IF VisitingExtension.Alarms.HasAlarms THEN
	serializer.addkey('alarms');
	serializer.StartArray();
	VisitingExtension.Alarms.Accept(THIS^);
	serializer.EndArray();
END_IF

IF VisitingExtension.InputPorts.HasInputPorts THEN
	serializer.addkey('inputPorts');
	serializer.StartArray();
	VisitingExtension.InputPorts.Accept(THIS^);
	serializer.EndArray();
END_IF

IF VisitingExtension.OutputPorts.HasOutputPorts THEN
	serializer.addkey('outputPorts');
	serializer.StartArray();
	VisitingExtension.OutputPorts.Accept(THIS^);
	serializer.EndArray();
END_IF

IF VisitingExtension.Parameters.HasParameters THEN
	serializer.addkey('parameters');
	serializer.StartArray();
	VisitingExtension.Parameters.Accept(THIS^);
	serializer.EndArray();
END_IF

IF VisitingExtension.Contents.HasContents THEN
	serializer.addkey('contents');
	serializer.StartArray();
	VisitingExtension.Contents.Accept(THIS^);
	serializer.EndArray();
END_IF

Serializer.EndObject();
END_METHOD

METHOD VisitInputPort
VAR_INPUT
	VisitingInputPort : I_InputPort;
END_VAR
serializer.StartObject();

serializer.AddKeyString('name', VisitingInputPort.Name);
serializer.Addkey('datatype');
VisitingInputPort.Data.SerializeTypeWith(serializer);

IF VisitingInputPort.Metadatum.HasMetadata THEN
	serializer.addkey('metadata');
	serializer.StartArray();
	VisitingInputPort.Metadatum.Accept(THIS^);
	serializer.EndArray();
END_IF

serializer.EndObject();
END_METHOD

METHOD VisitMetadatum
VAR_INPUT
	VisitingMetadatum : I_Metadata;
END_VAR
serializer.StartObject();
serializer.AddKeyString('name', VisitingMetadatum.Name);
serializer.AddkeyObject('value', VisitingMetadatum.Data);
serializer.EndObject();
END_METHOD

METHOD VisitNode
VAR_INPUT
	VisitingNode : I_Node;
END_VAR
serializer.StartObject();

IF VisitingNode.Metadatum.HasMetadata THEN
	serializer.addkey('metadata');
	serializer.StartArray();
	VisitingNode.Metadatum.Accept(THIS^);
	serializer.EndArray();
END_IF

IF VisitingNode.Alarms.HasAlarms THEN
	serializer.addkey('alarms');
	serializer.StartArray();
	VisitingNode.Alarms.Accept(THIS^);
	serializer.EndArray();
END_IF

IF VisitingNode.Extensions.HasExtensions THEN
	serializer.addkey('extensions');
	serializer.StartArray();
	VisitingNode.Extensions.Accept(THIS^);
	serializer.EndArray();
END_IF

IF VisitingNode.InputPorts.HasInputPorts THEN
	serializer.addkey('inputPorts');
	serializer.StartArray();
	VisitingNode.InputPorts.Accept(THIS^);
	serializer.EndArray();
END_IF

IF VisitingNode.OutputPorts.HasOutputPorts THEN
	serializer.addkey('outputPorts');
	serializer.StartArray();
	VisitingNode.OutputPorts.Accept(THIS^);
	serializer.EndArray();
END_IF

IF VisitingNode.Parameters.HasParameters THEN
	serializer.addkey('parameters');
	serializer.StartArray();
	VisitingNode.Parameters.Accept(THIS^);
	serializer.EndArray();
END_IF

IF VisitingNode.Contents.HasContents THEN
	serializer.addkey('contents');
	serializer.StartArray();
	VisitingNode.Contents.Accept(THIS^);
	serializer.EndArray();
END_IF

serializer.EndObject();
END_METHOD

METHOD VisitNodeFactory
VAR_INPUT
	VisitingNodeFactory : I_NodeFactory;
END_VAR
serializer.StartObject();
serializer.AddKey('blueprints');
serializer.StartArray();
VisitingNodeFactory.NodePrototypes.Accept(THIS^);
serializer.EndArray();
serializer.AddKeyUdint('returnedCount', blueprintsCollected);
serializer.AddKeyUdint('totalCount', totalBlueprints);
serializer.AddKeyUdint('nextOffset', offset + blueprintsCollected);
serializer.AddKeyBool('hasMore', offset + blueprintsCollected < totalBlueprints); 
serializer.EndObject();
END_METHOD

METHOD VisitNodePrototype
VAR_INPUT
	VisitingPrototype : I_NodePrototype;
END_VAR
// we're not yet in range of collection
IF currentIndex < offset THEN
	currentIndex := currentIndex + 1;
	totalBlueprints := totalBlueprints + 1;
	RETURN;
END_IF

// we're over range of the collection
IF currentIndex > endIndex THEN
	currentIndex := currentIndex + 1;
	totalBlueprints := totalBlueprints + 1;
	RETURN;
END_IF

// we're in the range to collect. 

blueprintsCollected := blueprintsCollected + 1;
currentIndex := currentIndex + 1;
totalBlueprints := totalBlueprints + 1;

serializer.StartObject();
serializer.AddKeyString('path', VisitingPrototype.Path);
serializer.AddKey('node');
VisitingPrototype.Node.Accept(THIS^);
serializer.EndObject();
END_METHOD

METHOD VisitOutputPort
VAR_INPUT
	VisitingOutputPort : I_OutputPort;
END_VAR
serializer.StartObject();

serializer.AddKeyString('name', VisitingOutputPort.Name);
serializer.Addkey('datatype');
VisitingOutputPort.Data.SerializeTypeWith(serializer);

IF VisitingOutputPort.Metadatum.HasMetadata THEN
	serializer.addkey('metadata');
	serializer.StartArray();
	VisitingOutputPort.Metadatum.Accept(THIS^);
	serializer.EndArray();
END_IF

serializer.EndObject();
END_METHOD

METHOD VisitParameter
VAR_INPUT
	VisitingProperty : I_Parameter;
END_VAR
serializer.StartObject();

serializer.AddKeyString('name', VisitingProperty.Name);
serializer.Addkey('datatype');
VisitingProperty.Data.SerializeTypeWith(serializer);
serializer.Addkey('defaultValue');
VisitingProperty.Data.SerializeWith(serializer);

IF VisitingProperty.Metadatum.HasMetadata THEN
	serializer.addkey('metadata');
	serializer.StartArray();
	VisitingProperty.Metadatum.Accept(THIS^);
	serializer.EndArray();
END_IF

Serializer.EndObject();
END_METHOD

END_FUNCTION_BLOCK

// API/Visitors/GetBlueprintsVisitor
{attribute 'linkalways'} 
{attribute 'no_explicit_call' := 'This FB is a CLASS and must be accessed using methods or properties'}
{attribute 'enable_dynamic_creation'}
FUNCTION_BLOCK GetBlueprintsVisitor IMPLEMENTS I_NodeFactoryVisitor, I_NodePrototypeVisitor, I_NodeVisitor, I_ExtensionVisitor, I_InputPortVisitor, I_OutputPortVisitor, I_MetadataVisitor, I_ContentVisitor, I_ParameterVisitor, I_AlarmVisitor
VAR
	serializer : I_Serializer;
END_VAR

METHOD PUBLIC Initialize
VAR_INPUT
	Serializer : I_Serializer;
END_VAR
THIS^.serializer := Serializer;
END_METHOD

METHOD VisitAlarm
VAR_INPUT
	VisitingAlarm : I_Alarm;
END_VAR
serializer.AddString(VisitingAlarm.Message);
END_METHOD

METHOD VisitContent
VAR_INPUT
	VisitingContent : I_Content;
END_VAR
serializer.StartObject();

serializer.AddKeyString('name', VisitingContent.Name);
serializer.Addkey('datatype');
VisitingContent.Data.SerializeTypeWith(serializer);

IF VisitingContent.Metadatum.HasMetadata THEN
	serializer.addkey('metadata');
	serializer.StartArray();
	VisitingContent.Metadatum.Accept(THIS^);
	serializer.EndArray();
END_IF

serializer.EndObject();
END_METHOD

METHOD VisitExtension
VAR_INPUT
	VisitingExtension : I_Extension;
END_VAR
Serializer.StartObject();
Serializer.AddKeyString('name', VisitingExtension.Name);

IF VisitingExtension.Metadatum.HasMetadata THEN
	serializer.addkey('metadata');
	serializer.StartArray();
	VisitingExtension.Metadatum.Accept(THIS^);
	serializer.EndArray();
END_IF

IF VisitingExtension.Alarms.HasAlarms THEN
	serializer.addkey('alarms');
	serializer.StartArray();
	VisitingExtension.Alarms.Accept(THIS^);
	serializer.EndArray();
END_IF

IF VisitingExtension.InputPorts.HasInputPorts THEN
	serializer.addkey('inputPorts');
	serializer.StartArray();
	VisitingExtension.InputPorts.Accept(THIS^);
	serializer.EndArray();
END_IF

IF VisitingExtension.OutputPorts.HasOutputPorts THEN
	serializer.addkey('outputPorts');
	serializer.StartArray();
	VisitingExtension.OutputPorts.Accept(THIS^);
	serializer.EndArray();
END_IF

IF VisitingExtension.Parameters.HasParameters THEN
	serializer.addkey('parameters');
	serializer.StartArray();
	VisitingExtension.Parameters.Accept(THIS^);
	serializer.EndArray();
END_IF

IF VisitingExtension.Contents.HasContents THEN
	serializer.addkey('contents');
	serializer.StartArray();
	VisitingExtension.Contents.Accept(THIS^);
	serializer.EndArray();
END_IF

Serializer.EndObject();
END_METHOD

METHOD VisitInputPort
VAR_INPUT
	VisitingInputPort : I_InputPort;
END_VAR
serializer.StartObject();

serializer.AddKeyString('name', VisitingInputPort.Name);
serializer.Addkey('datatype');
VisitingInputPort.Data.SerializeTypeWith(serializer);

IF VisitingInputPort.Metadatum.HasMetadata THEN
	serializer.addkey('metadata');
	serializer.StartArray();
	VisitingInputPort.Metadatum.Accept(THIS^);
	serializer.EndArray();
END_IF

serializer.EndObject();
END_METHOD

METHOD VisitMetadatum
VAR_INPUT
	VisitingMetadatum : I_Metadata;
END_VAR
serializer.StartObject();
serializer.AddKeyString('name', VisitingMetadatum.Name);
serializer.AddkeyObject('value', VisitingMetadatum.Data);
serializer.EndObject();
END_METHOD

METHOD VisitNode
VAR_INPUT
	VisitingNode : I_Node;
END_VAR
serializer.StartObject();

IF VisitingNode.Metadatum.HasMetadata THEN
	serializer.addkey('metadata');
	serializer.StartArray();
	VisitingNode.Metadatum.Accept(THIS^);
	serializer.EndArray();
END_IF

IF VisitingNode.Alarms.HasAlarms THEN
	serializer.addkey('alarms');
	serializer.StartArray();
	VisitingNode.Alarms.Accept(THIS^);
	serializer.EndArray();
END_IF

IF VisitingNode.Extensions.HasExtensions THEN
	serializer.addkey('extensions');
	serializer.StartArray();
	VisitingNode.Extensions.Accept(THIS^);
	serializer.EndArray();
END_IF

IF VisitingNode.InputPorts.HasInputPorts THEN
	serializer.addkey('inputPorts');
	serializer.StartArray();
	VisitingNode.InputPorts.Accept(THIS^);
	serializer.EndArray();
END_IF

IF VisitingNode.OutputPorts.HasOutputPorts THEN
	serializer.addkey('outputPorts');
	serializer.StartArray();
	VisitingNode.OutputPorts.Accept(THIS^);
	serializer.EndArray();
END_IF

IF VisitingNode.Parameters.HasParameters THEN
	serializer.addkey('parameters');
	serializer.StartArray();
	VisitingNode.Parameters.Accept(THIS^);
	serializer.EndArray();
END_IF

IF VisitingNode.Contents.HasContents THEN
	serializer.addkey('contents');
	serializer.StartArray();
	VisitingNode.Contents.Accept(THIS^);
	serializer.EndArray();
END_IF

serializer.EndObject();
END_METHOD

METHOD VisitNodeFactory
VAR_INPUT
	VisitingNodeFactory : I_NodeFactory;
END_VAR
serializer.StartObject();
serializer.AddKey('blueprints');
serializer.StartArray();
VisitingNodeFactory.NodePrototypes.Accept(THIS^);
serializer.EndArray();
serializer.EndObject();
END_METHOD

METHOD VisitNodePrototype
VAR_INPUT
	VisitingPrototype : I_NodePrototype;
END_VAR
serializer.StartObject();
serializer.AddKeyString('path', VisitingPrototype.Path);
serializer.AddKey('node');
VisitingPrototype.Node.Accept(THIS^);
serializer.EndObject();
END_METHOD

METHOD VisitOutputPort
VAR_INPUT
	VisitingOutputPort : I_OutputPort;
END_VAR
serializer.StartObject();

serializer.AddKeyString('name', VisitingOutputPort.Name);
serializer.Addkey('datatype');
VisitingOutputPort.Data.SerializeTypeWith(serializer);

IF VisitingOutputPort.Metadatum.HasMetadata THEN
	serializer.addkey('metadata');
	serializer.StartArray();
	VisitingOutputPort.Metadatum.Accept(THIS^);
	serializer.EndArray();
END_IF

serializer.EndObject();
END_METHOD

METHOD VisitParameter
VAR_INPUT
	VisitingProperty : I_Parameter;
END_VAR
serializer.StartObject();

serializer.AddKeyString('name', VisitingProperty.Name);
serializer.Addkey('datatype');
VisitingProperty.Data.SerializeTypeWith(serializer);
serializer.Addkey('defaultValue');
VisitingProperty.Data.SerializeWith(serializer);

IF VisitingProperty.Metadatum.HasMetadata THEN
	serializer.addkey('metadata');
	serializer.StartArray();
	VisitingProperty.Metadatum.Accept(THIS^);
	serializer.EndArray();
END_IF

Serializer.EndObject();
END_METHOD

END_FUNCTION_BLOCK

// API/Handlers/GetContentValueHandler
{attribute 'linkalways'} 
{attribute 'no_explicit_call' := 'This FB is a CLASS and must be accessed using methods or properties'}
{attribute 'enable_dynamic_creation'}
FUNCTION_BLOCK GetContentValueHandler IMPLEMENTS I_AsynchronousRpcHandler
VAR
	graphRuntimes : I_GraphRuntimeCollection;
END_VAR

METHOD Handle
VAR_INPUT
	Parameters : I_Deserializer;
	Response : I_AsynchronousRpcResponse;
END_VAR
VAR
	runtimeId : T_MAXSTRING;
	graphRuntime : I_GraphRuntime;
	graphInstanceId : T_MAXSTRING;
	graphInstance : I_GraphInstance;
	graphUuid : T_MAXSTRING;
	nodeId : T_MAXSTRING;
	contentName : T_MAXSTRING;
	visitor : RetrieveNodeContentValue;
	serializer : I_Serializer;
	feedback : DeserializerFeedback;
END_VAR
IF graphRuntimes = 0 THEN
	Response.RejectWithError('INTERNAL_ERROR','GetContentValueHandler has not been correctly initialized');
	RETURN;
END_IF

// get runtime
IF Parameters.TryGetKeyString('runtimeId', runtimeId, feedback) THEN
	IF NOT graphRuntimes.TryGetRuntimeById(runtimeId, graphRuntime) THEN
		Response.RejectWithError('INVALID_RUNTIME_ID','The runtimeId is missing or invalid');
		RETURN;
	END_IF
ELSE
	IF NOT graphRuntimes.TryGetDefaultRuntime(graphRuntime) THEN
		Response.RejectWithError('INTERNAL_ERROR','Unable to get default runtime');
		RETURN;
	END_IF
END_IF

// get graph instance
IF Parameters.TryGetKeyString('graphInstanceId', graphInstanceId, feedback) THEN
	IF NOT graphRuntime.TryGetGraphInstance(graphInstanceId, graphInstance) THEN
		Response.RejectWithError('INVALID_GRAPH_INSTANCE_ID','The graphInstanceId is missing or invalid');
		RETURN;
	END_IF
ELSE
	IF NOT graphRuntime.TryGetDefaultGraphInstance(graphInstance) THEN
		Response.RejectWithError('NO_GRAPH_INSTANCE_AVAILABLE','Unable to get default graph instance, i.e. no graph instance is loaded');
		RETURN;
	END_IF
END_IF

// setup the visitor
IF NOT Parameters.TryGetKeyString('graphUuid', graphUuid, feedback) THEN
	Response.RejectWithError('MISSING_GRAPH_UUID_PARAMETER',feedback.FirstError.Message);
	RETURN;
END_IF

IF NOT (graphUuid = graphInstance.Graph.Uuid) THEN
	Response.RejectWithError('GRAPH_UUID_MISSMATCH','The requested uuid did not match the graph instance found');
	RETURN;
END_IF

IF NOT Parameters.TryGetKeyString('nodeId', nodeId, feedback) THEN
	Response.RejectWithError('MISSING_NODE_ID_PARAMETER',feedback.FirstError.Message);
	RETURN;
END_IF

IF NOT Parameters.TryGetKeyString('contentName', contentName, feedback) THEN
	Response.RejectWithError('MISSING_CONTENT_NAME_PARAMETER',feedback.FirstError.Message);
	RETURN;
END_IF

serializer := Response.GetSerializer();
visitor.Initialize(graphUuid, nodeId, contentName, serializer);
graphInstance.graph.Accept(visitor);

IF visitor.Error THEN
	Response.RejectWithError('GET_CONTENT_FAILED',visitor.ErrorMessage);
	serializer.Dispose();
	RETURN;
END_IF

IF NOT visitor.Done THEN
	Response.RejectWithError('GET_CONTENT_FAILED','Unable to get content from graph');
	serializer.Dispose();
	RETURN;
END_IF

Response.CompleteWithSerializer(serializer);
serializer.Dispose();
END_METHOD

METHOD PUBLIC Initialize
VAR_INPUT
	GraphRuntimes : I_GraphRuntimeCollection;
END_VAR
THIS^.graphRuntimes := GraphRuntimes;
END_METHOD

END_FUNCTION_BLOCK

// API/Visitors/RetrieveNodeContentValue
{attribute 'linkalways'} 
{attribute 'no_explicit_call' := 'This FB is a CLASS and must be accessed using methods or properties'}
{attribute 'enable_dynamic_creation'}
FUNCTION_BLOCK RetrieveNodeContentValue IMPLEMENTS I_GraphVisitor, I_NodeVisitor, I_ContentVisitor
VAR
	graphUuid : T_MAXSTRING;
	nodeId : T_MAXSTRING;
	contentName : T_MAXSTRING;
	serializer : I_Serializer;
	_done : BOOL;
	_error : BOOL;
	_errorMessage : T_MAXSTRING;
END_VAR

METHOD PRIVATE LogInvalidContentNameError
VAR_INPUT
END_VAR
_errorMessage := 'Invalid Content Name';
_error := TRUE;
END_METHOD

METHOD PRIVATE LogInvalidNodeIdError
VAR_INPUT
END_VAR
_errorMessage := 'Invalid Node Id';
_error := TRUE;
END_METHOD

METHOD PRIVATE Reset
VAR_INPUT
END_VAR
_done := FALSE;
_errorMessage := '';
_error := FALSE;
END_METHOD

PROPERTY PUBLIC Done : BOOL
GET
Done := _done;
END_GET
END_PROPERTY

PROPERTY PUBLIC Error : BOOL
GET
Error := _error;
END_GET
END_PROPERTY

PROPERTY PUBLIC ErrorMessage : T_MAXSTRING
GET
ErrorMessage := _errorMessage;
END_GET
END_PROPERTY

METHOD PUBLIC Initialize
VAR_INPUT
	GraphUuid : T_MAXSTRING;
	NodeId : T_MAXSTRING;
	ContentName : T_MAXSTRING;
	Serializer : I_Serializer;
END_VAR
THIS^.graphUuid := GraphUuid;
THIS^.nodeId := NodeId;
THIS^.contentName := ContentName;
THIS^.serializer := Serializer;
END_METHOD

METHOD VisitContent
VAR_INPUT
	VisitingContent : I_Content;
END_VAR
VisitingContent.SerializeWith(serializer);
END_METHOD

METHOD VisitGraph
VAR_INPUT
	VisitingGraph : I_Graph;
END_VAR
VAR
	node : I_Node;
END_VAR
Reset();

IF NOT (VisitingGraph.Uuid = graphUuid) THEN
	RETURN;
END_IF

IF NOT VisitingGraph.Nodes.TryGetNodeById(nodeId, node) THEN
	LogInvalidNodeIdError();
	RETURN;
END_IF

node.Accept(THIS^);
END_METHOD

METHOD VisitNode
VAR_INPUT
	VisitingNode : I_Node;
END_VAR
VAR
	content : I_Content;
END_VAR
IF NOT VisitingNode.Contents.TryGetContentByName(contentName, content) THEN
	LogInvalidContentNameError();
	RETURN;
END_IF

content.Accept(THIS^);
END_METHOD

END_FUNCTION_BLOCK

// API/Handlers/GetStatusRpcHandler
{attribute 'linkalways'} 
{attribute 'no_explicit_call' := 'This FB is a CLASS and must be accessed using methods or properties'}
{attribute 'enable_dynamic_creation'}
FUNCTION_BLOCK GetStatusRpcHandler IMPLEMENTS I_AsynchronousRpcHandler
VAR
	graphRuntimes : I_GraphRuntimeCollection;
END_VAR

METHOD Handle
VAR_INPUT
	Parameters : I_Deserializer;
	Response : I_AsynchronousRpcResponse;
END_VAR
VAR
	runtimeId : T_MAXSTRING;
	graphRuntime : I_GraphRuntime;
	graphInstanceId : T_MAXSTRING;
	graphUuid : T_MAXSTRING;
	graphInstance : I_GraphInstance;
	feedback : DeserializerFeedback;
	serializer : I_Serializer;
	getStatusVisitor : GetStatusVisitor;
END_VAR
IF graphRuntimes = 0 THEN
	Response.RejectWithError('INTERNAL_ERROR','GetStatusRpcHandler has not been correctly initialized');
	RETURN;
END_IF

// get runtime
IF Parameters.TryGetKeyString('runtimeId', runtimeId, feedback) THEN
	IF NOT graphRuntimes.TryGetRuntimeById(runtimeId, graphRuntime) THEN
		Response.RejectWithError('INVALID_RUNTIME_ID','The runtimeId is missing or invalid');
		RETURN;
	END_IF
ELSE
	IF NOT graphRuntimes.TryGetDefaultRuntime(graphRuntime) THEN
		Response.RejectWithError('INTERNAL_ERROR','Unable to get default runtime');
		RETURN;
	END_IF
END_IF

// get graph instance
IF Parameters.TryGetKeyString('graphInstanceId', graphInstanceId, feedback) THEN
	IF NOT graphRuntime.TryGetGraphInstance(graphInstanceId, graphInstance) THEN
		Response.RejectWithError('INVALID_GRAPH_INSTANCE_ID','The graphInstanceId is missing or invalid');
		RETURN;
	END_IF
ELSE
	IF NOT graphRuntime.TryGetDefaultGraphInstance(graphInstance) THEN
		Response.RejectWithError('NO_GRAPH_INSTANCE_AVAILABLE','Unable to get default graph instance, i.e. no graph instance is loaded');
		RETURN;
	END_IF
END_IF

// setup the visitor
IF NOT Parameters.TryGetKeyString('graphUuid', graphUuid, feedback) THEN
	Response.RejectWithError('MISSING_GRAPH_UUID_PARAMETER', feedback.FirstError.Message);
	RETURN;
END_IF

IF NOT (graphUuid = graphInstance.Graph.Uuid) THEN
	Response.RejectWithError('GRAPH_UUID_MISSMATCH','The requested uuid did not match the graph instance found');
	RETURN;
END_IF

serializer := Response.GetSerializer();
getStatusVisitor.Initialize(serializer);
getStatusVisitor.VisitGraph(graphInstance.Graph);
Response.CompleteWithSerializer(serializer);
serializer.Dispose();
END_METHOD

METHOD PUBLIC Initialize
VAR_INPUT
	GraphRuntimes : I_GraphRuntimeCollection;
END_VAR
THIS^.graphRuntimes := GraphRuntimes;
END_METHOD

END_FUNCTION_BLOCK

// API/Handlers/UpdateParameterValueHandler
{attribute 'linkalways'} 
{attribute 'no_explicit_call' := 'This FB is a CLASS and must be accessed using methods or properties'}
{attribute 'enable_dynamic_creation'}
FUNCTION_BLOCK UpdateParameterValueHandler IMPLEMENTS I_AsynchronousRpcHandler
VAR
	graphRuntimes : I_GraphRuntimeCollection;
END_VAR

METHOD Handle
VAR_INPUT
	Parameters : I_Deserializer;
	Response : I_AsynchronousRpcResponse;
END_VAR
VAR
	runtimeId : T_MAXSTRING;
	graphRuntime : I_GraphRuntime;
	graphInstanceId : T_MAXSTRING;
	graphUuid : T_MAXSTRING;
	graphInstance : I_GraphInstance;
	nodeId : T_MAXSTRING;
	node : I_Node;
	parameterName : T_MAXSTRING;
	parameter : I_Parameter;
	visitor : RetrieveNodeContentValue;
	serializer : I_Serializer;
	feedback : DeserializerFeedback;
END_VAR
IF graphRuntimes = 0 THEN
	Response.RejectWithError('INTERNAL_ERROR','UpdateParameterValueHandler has not been correctly initialized');
	RETURN;
END_IF

// get runtime
IF Parameters.TryGetKeyString('runtimeId', runtimeId, feedback) THEN
	IF NOT graphRuntimes.TryGetRuntimeById(runtimeId, graphRuntime) THEN
		Response.RejectWithError('INVALID_RUNTIME_ID','The runtimeId is missing or invalid');
		RETURN;
	END_IF
ELSE
	IF NOT graphRuntimes.TryGetDefaultRuntime(graphRuntime) THEN
		Response.RejectWithError('INTERNAL_ERROR','Unable to get default runtime');
		RETURN;
	END_IF
END_IF

// get graph instance
IF Parameters.TryGetKeyString('graphInstanceId', graphInstanceId, feedback) THEN
	IF NOT graphRuntime.TryGetGraphInstance(graphInstanceId, graphInstance) THEN
		Response.RejectWithError('INVALID_GRAPH_INSTANCE_ID','The graphInstanceId is missing or invalid');
		RETURN;
	END_IF
ELSE
	IF NOT graphRuntime.TryGetDefaultGraphInstance(graphInstance) THEN
		Response.RejectWithError('NO_GRAPH_INSTANCE_AVAILABLE','Unable to get default graph instance, i.e. no graph instance is loaded');
		RETURN;
	END_IF
END_IF

// setup the visitor
IF NOT Parameters.TryGetKeyString('graphUuid', graphUuid, feedback) THEN
	Response.RejectWithError('MISSING_GRAPH_UUID_PARAMETER',feedback.FirstError.Message);
	RETURN;
END_IF

IF NOT (graphUuid = graphInstance.Graph.Uuid) THEN
	Response.RejectWithError('GRAPH_UUID_MISSMATCH', 'The requested uuid did not match the graph instance found');
	RETURN;
END_IF

IF NOT Parameters.TryGetKeyString('nodeId', nodeId, feedback) THEN
	Response.RejectWithError('MISSING_NODE_ID_PARAMETER',feedback.FirstError.Message);
	RETURN;
END_IF

IF NOT graphInstance.Graph.Nodes.TryGetNodeById(nodeId, node) THEN
	Response.RejectWithError('INVALID_NODE_ID','Invalid or missing nodeId');
	RETURN;
END_IF

IF NOT Parameters.TryGetKeyString('parameterName', parameterName, feedback) THEN
	Response.RejectWithError('MISSING_PARAMETER_NAME_PARAMETER',feedback.FirstError.Message);
	RETURN;
END_IF

IF NOT node.Parameters.TryGetParameterByName(parameterName, parameter) THEN
	Response.RejectWithError('INVALID_PARAMETER_NAME','Invalid or missing parameterName');
	RETURN;
END_IF

IF NOT Parameters.TryDeserializeKeyToObject ('parameterValue', parameter, feedback) THEN
	Response.RejectWithError('MISSING_PARAMETER_VALUE_PARAMETER',feedback.FirstError.Message);
	RETURN;
END_IF

Response.CompleteWithString(graphUuid);
END_METHOD

METHOD PUBLIC Initialize
VAR_INPUT
	GraphRuntimes : I_GraphRuntimeCollection;
END_VAR
THIS^.graphRuntimes := GraphRuntimes;
END_METHOD

END_FUNCTION_BLOCK

// API/GraphFrameworkApi
{attribute 'linkalways'} 
{attribute 'no_explicit_call' := 'This FB is a CLASS and must be accessed using methods or properties'}
{attribute 'enable_dynamic_creation'}
FUNCTION_BLOCK GraphFrameworkApi IMPLEMENTS I_RpcApi
VAR
	graphFramework : I_GraphFramework;
	graphRuntimes : GraphRuntimeCollection;
	createGraphRpcHandler : CreateGraphRpcHandler;
	getStatusRpcHandler : GetStatusRpcHandler;
	getBlueprintsRpcHandler : GetBlueprintsRpcHandler;
	getContentValueHandler : GetContentValueHandler;
	updateParameterValueHandler : UpdateParameterValueHandler;
END_VAR

METHOD FB_init : BOOL
VAR_INPUT
	bInitRetains : BOOL; // if TRUE, the retain variables are initialized (warm start / cold start)
	bInCopyCode : BOOL;  // if TRUE, the instance afterwards gets moved into the copy code (online change)
	GraphFramework : I_GraphFramework;
	DefaultGraphRuntime : I_GraphRuntime;
END_VAR
THIS^.graphFramework := GraphFramework;
THIS^.graphRuntimes.AddDefaultRuntime(DefaultGraphRuntime);

getBlueprintsRpcHandler.Initialize(GraphFramework);
getStatusRpcHandler.Initialize(graphRuntimes);
createGraphRpcHandler.Initialize(GraphFramework, graphRuntimes);
getContentValueHandler.Initialize(graphRuntimes);
updateParameterValueHandler.Initialize(graphRuntimes);
END_METHOD

METHOD PUBLIC AddRuntimeById
VAR_INPUT
	Id : T_MAXSTRING;
	GraphRuntime : I_GraphRuntime;
END_VAR
graphRuntimes.AddRuntimeById(Id, GraphRuntime);
END_METHOD

METHOD CyclicCall
VAR_INPUT
END_VAR
// no implementation
END_METHOD

METHOD RegisterAsynchronousRpcHandlersWith
VAR_INPUT
	Host : I_HostAsynchronousRpcHandlers;
END_VAR
Host.RegisterHandler('CreateGraph', createGraphRpcHandler);
Host.RegisterHandler('GetStatus', getStatusRpcHandler);
Host.RegisterHandler('GetBlueprints', getBlueprintsRpcHandler);
Host.RegisterHandler('GetContentValue', getContentValueHandler);
Host.RegisterHandler('UpdateParameterValue', updateParameterValueHandler);
END_METHOD

METHOD RegisterSynchronousRpcHandlersWith
VAR_INPUT
	Host : I_HostSynchronousRpcHandlers;
END_VAR
// no implementation
END_METHOD

END_FUNCTION_BLOCK

// GraphRuntime/Collection/GraphRuntimeCollection
{attribute 'linkalways'} 
{attribute 'no_explicit_call' := 'This FB is a CLASS and must be accessed using methods or properties'}
{attribute 'enable_dynamic_creation'}
FUNCTION_BLOCK GraphRuntimeCollection IMPLEMENTS I_GraphRuntimeCollection
VAR
	graphRuntimes : Dictionary;
	enumerator : I_ForwardEnumerator;
END_VAR
VAR CONSTANT
	DEFAULT_ID : T_MAXSTRING := 'default';
END_VAR

METHOD FB_init : BOOL
VAR_INPUT
	bInitRetains : BOOL; // if TRUE, the retain variables are initialized (warm start / cold start)
	bInCopyCode : BOOL;  // if TRUE, the instance afterwards gets moved into the copy code (online change)
END_VAR
GetNewEnumerator();
END_METHOD

METHOD FB_exit : BOOL
VAR_INPUT
	bInCopyCode : BOOL; // if TRUE, the exit method is called for exiting an instance that is copied afterwards (online change).
END_VAR
DisposeEnumerator();
END_METHOD

METHOD PRIVATE DisposeEnumerator
VAR_INPUT
END_VAR
IF enumerator = 0 THEN
	RETURN;
END_IF

enumerator.Dispose();
enumerator := 0;
END_METHOD

METHOD PRIVATE GetNewEnumerator
VAR_INPUT
END_VAR
IF enumerator <> 0 THEN
	enumerator.Dispose();
	enumerator := 0;
END_IF

enumerator := graphRuntimes.GetEnumerator();
END_METHOD

METHOD PUBLIC Accept
VAR_INPUT
	visitor : I_GraphRuntimeVisitor;
END_VAR
VAR
	graphRuntime : I_GraphRuntime;
END_VAR
IF NOT enumerator.IsValid THEN
	GetNewEnumerator();
ELSE
	enumerator.Reset();
END_IF

WHILE (enumerator.MoveNext()) DO
	
	IF enumerator.TryGet(graphRuntime) THEN
		graphRuntime.Accept(Visitor);
	END_IF

END_WHILE
END_METHOD

METHOD PUBLIC AddDefaultRuntime
VAR_INPUT
	GraphRuntime : I_GraphRuntime;
END_VAR
AddRuntimeById(DEFAULT_ID, GraphRuntime);
END_METHOD

METHOD PUBLIC AddRuntimeById
VAR_INPUT
	Id : T_MAXSTRING;
	GraphRuntime : I_GraphRuntime;
END_VAR
IF GraphRuntime = 0 THEN
	RETURN;
END_IF

graphRuntimes.AddOrUpdate(Id, GraphRuntime);
END_METHOD

METHOD PUBLIC RemoveDefaultRuntime
VAR_INPUT
END_VAR
RemoveRuntimeById(DEFAULT_ID);
END_METHOD

METHOD PUBLIC RemoveRuntimeById
VAR_INPUT
	Id : T_MAXSTRING;
END_VAR
graphRuntimes.Remove(Id);
END_METHOD

METHOD PUBLIC TryGetDefaultRuntime : BOOL
VAR_INPUT
	Destination : REFERENCE TO I_GraphRuntime;
END_VAR
TryGetDefaultRuntime := TryGetRuntimeById(DEFAULT_ID, Destination);
END_METHOD

METHOD PUBLIC TryGetRuntimeById : BOOL
VAR_INPUT
	Id : T_MAXSTRING;
	Destination : REFERENCE TO I_GraphRuntime;
END_VAR
VAR
	graphRuntime : I_GraphRuntime;
END_VAR
IF NOT graphRuntimes.TryGetValue(Id, graphRuntime) THEN
	RETURN;
END_IF

Destination := graphRuntime;
TryGetRuntimeById := TRUE;
END_METHOD

END_FUNCTION_BLOCK

// Extensions/Namespace/ExtensionNamespace
{attribute 'linkalways'} 
{attribute 'no_explicit_call' := 'This FB is a CLASS and must be accessed using methods or properties'}
{attribute 'enable_dynamic_creation'}
FUNCTION_BLOCK ExtensionNamespace
VAR
	_extensionName : T_MAXSTRING;
	_targetName : T_MAXSTRING;
	_isExtensionPath : BOOL;
END_VAR

METHOD FB_init : BOOL
VAR_INPUT
	bInitRetains : BOOL; // if TRUE, the retain variables are initialized (warm start / cold start)
	bInCopyCode : BOOL;  // if TRUE, the instance afterwards gets moved into the copy code (online change)
	Path : T_MAXSTRING;
END_VAR
Initialize(Path);
END_METHOD

PROPERTY PUBLIC ExtensionName : T_MAXSTRING
GET
IF NOT _isExtensionPath THEN
	RETURN;
END_IF

ExtensionName := _extensionNAme;
END_GET
END_PROPERTY

METHOD PUBLIC Initialize
VAR_INPUT
	Path : T_MAXSTRING;
END_VAR
_isExtensionPath := FindAndSplitChar(
	sSeparatorChar := '.',  
	pSrcString := ADR(Path),                                  
	pLeftString := ADR(_extensionName),   
	nLeftSize := SIZEOF(_extensionName),                                  
	pRightString := ADR(_targetName), 
	nRightSize := SIZEOF(_targetName),                                
	bSearchFromRight := TRUE 
);
END_METHOD

PROPERTY PUBLIC IsExtensionPath : BOOL
GET
IsExtensionPath := _isExtensionPath;
END_GET
END_PROPERTY

PROPERTY PUBLIC TargetName : T_MAXSTRING
GET
IF NOT _isExtensionPath THEN
	RETURN;
END_IF

TargetName := _targetName;
END_GET
END_PROPERTY

END_FUNCTION_BLOCK

// IecDatatypesPack/IecDatatypesPack
{attribute 'linkalways'} 
{attribute 'no_explicit_call' := 'This FB is a CLASS and must be accessed using methods or properties'}
{attribute 'enable_dynamic_creation'}
FUNCTION_BLOCK IecDatatypesPack IMPLEMENTS I_GraphPack
VAR
	// _bit not included as this can only be part of a structure
	_bool : _BOOL(FALSE);
	_byte : _BYTE(0);
	_dint : _DINT(0);
	_dt : _DT(DT#1970-1-1-0:0:0);
	_dword : _DWORD(0);
	_int : _INT(0);
	_lint : _LINT(0);
	_lreal : _LREAL(0);
	_lword : _LWORD(0);
	_real : _REAL(0);
	_sint : _SINT(0);
	_time_of_day : _TIME_OF_DAY(TOD#0:0:0);
	_tod : _TOD(TOD#0:0:0);
	_udint : _UDINT(0);
	_uint : _UINT(0);
	_ulint : _ULINT(0);
	_usint : _USINT(0);
	_word : _WORD(0);
    _string : _STRING('');
	_pvoid : _PVOID;
	
	// converters
	
	// _to_bool
	_bool_to_bool_ConverterNode : ConverterNode(_bool, _bool);
	_byte_to_bool_ConverterNode : ConverterNode(_byte, _bool);
	_dint_to_bool_ConverterNode : ConverterNode(_dint, _bool);
	_dt_to_bool_ConverterNode : ConverterNode(_dt, _bool);
	_dword_to_bool_ConverterNode : ConverterNode(_dword, _bool);
	_int_to_bool_ConverterNode : ConverterNode(_int, _bool);
	_lint_to_bool_ConverterNode : ConverterNode(_lint, _bool);
	_lreal_to_bool_ConverterNode : ConverterNode(_lreal, _bool);
	_lword_to_bool_ConverterNode : ConverterNode(_lword, _bool);
	_real_to_bool_ConverterNode : ConverterNode(_real, _bool);
	_sint_to_bool_ConverterNode : ConverterNode(_sint, _bool);
	_tod_to_bool_ConverterNode : ConverterNode(_tod, _bool);
	_udint_to_bool_ConverterNode : ConverterNode(_udint, _bool);
	_uint_to_bool_ConverterNode : ConverterNode(_uint, _bool);
	_ulint_to_bool_ConverterNode : ConverterNode(_ulint, _bool);
	_usint_to_bool_ConverterNode : ConverterNode(_usint, _bool);
	_word_to_bool_ConverterNode : ConverterNode(_word, _bool);
	_string_to_bool_ConverterNode : ConverterNode(_string, _bool);
	_bool_to_byte_ConverterNode : ConverterNode(_bool, _byte);
	
	// _to_byte
	_byte_to_byte_ConverterNode : ConverterNode(_byte, _byte);
	_dint_to_byte_ConverterNode : ConverterNode(_dint, _byte);
	_dt_to_byte_ConverterNode : ConverterNode(_dt, _byte);
	_dword_to_byte_ConverterNode : ConverterNode(_dword, _byte);
	_int_to_byte_ConverterNode : ConverterNode(_int, _byte);
	_lint_to_byte_ConverterNode : ConverterNode(_lint, _byte);
	_lreal_to_byte_ConverterNode : ConverterNode(_lreal, _byte);
	_lword_to_byte_ConverterNode : ConverterNode(_lword, _byte);
	_real_to_byte_ConverterNode : ConverterNode(_real, _byte);
	_sint_to_byte_ConverterNode : ConverterNode(_sint, _byte);
	_tod_to_byte_ConverterNode : ConverterNode(_tod, _byte);
	_udint_to_byte_ConverterNode : ConverterNode(_udint, _byte);
	_uint_to_byte_ConverterNode : ConverterNode(_uint, _byte);
	_ulint_to_byte_ConverterNode : ConverterNode(_ulint, _byte);
	_usint_to_byte_ConverterNode : ConverterNode(_usint, _byte);
	_word_to_byte_ConverterNode : ConverterNode(_word, _byte);
	_string_to_byte_ConverterNode : ConverterNode(_string, _byte);

	// _to_dint
	_bool_to_dint_ConverterNode : ConverterNode(_bool, _dint);
	_byte_to_dint_ConverterNode : ConverterNode(_byte, _dint);
	_dint_to_dint_ConverterNode : ConverterNode(_dint, _dint);
	_dt_to_dint_ConverterNode : ConverterNode(_dt, _dint);
	_dword_to_dint_ConverterNode : ConverterNode(_dword, _dint);
	_int_to_dint_ConverterNode : ConverterNode(_int, _dint);
	_lint_to_dint_ConverterNode : ConverterNode(_lint, _dint);
	_lreal_to_dint_ConverterNode : ConverterNode(_lreal, _dint);
	_lword_to_dint_ConverterNode : ConverterNode(_lword, _dint);
	_real_to_dint_ConverterNode : ConverterNode(_real, _dint);
	_sint_to_dint_ConverterNode : ConverterNode(_sint, _dint);
	_tod_to_dint_ConverterNode : ConverterNode(_tod, _dint);
	_udint_to_dint_ConverterNode : ConverterNode(_udint, _dint);
	_uint_to_dint_ConverterNode : ConverterNode(_uint, _dint);
	_ulint_to_dint_ConverterNode : ConverterNode(_ulint, _dint);
	_usint_to_dint_ConverterNode : ConverterNode(_usint, _dint);
	_word_to_dint_ConverterNode : ConverterNode(_word, _dint);
	_string_to_dint_ConverterNode : ConverterNode(_string, _dint);

	// _to_dt
	_bool_to_dt_ConverterNode : ConverterNode(_bool, _dt);
	_byte_to_dt_ConverterNode : ConverterNode(_byte, _dt);
	_dint_to_dt_ConverterNode : ConverterNode(_dint, _dt);
	_dt_to_dt_ConverterNode : ConverterNode(_dt, _dt);
	_dword_to_dt_ConverterNode : ConverterNode(_dword, _dt);
	_int_to_dt_ConverterNode : ConverterNode(_int, _dt);
	_lint_to_dt_ConverterNode : ConverterNode(_lint, _dt);
	_lreal_to_dt_ConverterNode : ConverterNode(_lreal, _dt);
	_lword_to_dt_ConverterNode : ConverterNode(_lword, _dt);
	_real_to_dt_ConverterNode : ConverterNode(_real, _dt);
	_sint_to_dt_ConverterNode : ConverterNode(_sint, _dt);
	_tod_to_dt_ConverterNode : ConverterNode(_tod, _dt);
	_udint_to_dt_ConverterNode : ConverterNode(_udint, _dt);
	_uint_to_dt_ConverterNode : ConverterNode(_uint, _dt);
	_ulint_to_dt_ConverterNode : ConverterNode(_ulint, _dt);
	_usint_to_dt_ConverterNode : ConverterNode(_usint, _dt);
	_word_to_dt_ConverterNode : ConverterNode(_word, _dt);
	_string_to_dt_ConverterNode : ConverterNode(_string, _dt);

	// _to_dword
	_bool_to_dword_ConverterNode : ConverterNode(_bool, _dword);
	_byte_to_dword_ConverterNode : ConverterNode(_byte, _dword);
	_dint_to_dword_ConverterNode : ConverterNode(_dint, _dword);
	_dt_to_dword_ConverterNode : ConverterNode(_dt, _dword);
	_dword_to_dword_ConverterNode : ConverterNode(_dword, _dword);
	_int_to_dword_ConverterNode : ConverterNode(_int, _dword);
	_lint_to_dword_ConverterNode : ConverterNode(_lint, _dword);
	_lreal_to_dword_ConverterNode : ConverterNode(_lreal, _dword);
	_lword_to_dword_ConverterNode : ConverterNode(_lword, _dword);
	_real_to_dword_ConverterNode : ConverterNode(_real, _dword);
	_sint_to_dword_ConverterNode : ConverterNode(_sint, _dword);
	_tod_to_dword_ConverterNode : ConverterNode(_tod, _dword);
	_udint_to_dword_ConverterNode : ConverterNode(_udint, _dword);
	_uint_to_dword_ConverterNode : ConverterNode(_uint, _dword);
	_ulint_to_dword_ConverterNode : ConverterNode(_ulint, _dword);
	_usint_to_dword_ConverterNode : ConverterNode(_usint, _dword);
	_word_to_dword_ConverterNode : ConverterNode(_word, _dword);
	_string_to_dword_ConverterNode : ConverterNode(_string, _dword);
	
	// _to_int
	_bool_to_int_ConverterNode : ConverterNode(_bool, _int);
	_byte_to_int_ConverterNode : ConverterNode(_byte, _int);
	_dint_to_int_ConverterNode : ConverterNode(_dint, _int);
	_dt_to_int_ConverterNode : ConverterNode(_dt, _int);
	_dword_to_int_ConverterNode : ConverterNode(_dword, _int);
	_int_to_int_ConverterNode : ConverterNode(_int, _int);
	_lint_to_int_ConverterNode : ConverterNode(_lint, _int);
	_lreal_to_int_ConverterNode : ConverterNode(_lreal, _int);
	_lword_to_int_ConverterNode : ConverterNode(_lword, _int);
	_real_to_int_ConverterNode : ConverterNode(_real, _int);
	_sint_to_int_ConverterNode : ConverterNode(_sint, _int);
	_tod_to_int_ConverterNode : ConverterNode(_tod, _int);
	_udint_to_int_ConverterNode : ConverterNode(_udint, _int);
	_uint_to_int_ConverterNode : ConverterNode(_uint, _int);
	_ulint_to_int_ConverterNode : ConverterNode(_ulint, _int);
	_usint_to_int_ConverterNode : ConverterNode(_usint, _int);
	_word_to_int_ConverterNode : ConverterNode(_word, _int);
	_string_to_int_ConverterNode : ConverterNode(_string, _int);
	
	// _to_lint
	_bool_to_lint_ConverterNode : ConverterNode(_bool, _lint);
	_byte_to_lint_ConverterNode : ConverterNode(_byte, _lint);
	_dint_to_lint_ConverterNode : ConverterNode(_dint, _lint);
	_dt_to_lint_ConverterNode : ConverterNode(_dt, _lint);
	_dword_to_lint_ConverterNode : ConverterNode(_dword, _lint);
	_int_to_lint_ConverterNode : ConverterNode(_int, _lint);
	_lint_to_lint_ConverterNode : ConverterNode(_lint, _lint);
	_lreal_to_lint_ConverterNode : ConverterNode(_lreal, _lint);
	_lword_to_lint_ConverterNode : ConverterNode(_lword, _lint);
	_real_to_lint_ConverterNode : ConverterNode(_real, _lint);
	_sint_to_lint_ConverterNode : ConverterNode(_sint, _lint);
	_tod_to_lint_ConverterNode : ConverterNode(_tod, _lint);
	_udint_to_lint_ConverterNode : ConverterNode(_udint, _lint);
	_uint_to_lint_ConverterNode : ConverterNode(_uint, _lint);
	_ulint_to_lint_ConverterNode : ConverterNode(_ulint, _lint);
	_usint_to_lint_ConverterNode : ConverterNode(_usint, _lint);
	_word_to_lint_ConverterNode : ConverterNode(_word, _lint);
	_string_to_lint_ConverterNode : ConverterNode(_string, _lint);
	
	// _to_lreal
	_bool_to_lreal_ConverterNode : ConverterNode(_bool, _lreal);
	_byte_to_lreal_ConverterNode : ConverterNode(_byte, _lreal);
	_dint_to_lreal_ConverterNode : ConverterNode(_dint, _lreal);
	_dt_to_lreal_ConverterNode : ConverterNode(_dt, _lreal);
	_dword_to_lreal_ConverterNode : ConverterNode(_dword, _lreal);
	_int_to_lreal_ConverterNode : ConverterNode(_int, _lreal);
	_lint_to_lreal_ConverterNode : ConverterNode(_lint, _lreal);
	_lreal_to_lreal_ConverterNode : ConverterNode(_lreal, _lreal);
	_lword_to_lreal_ConverterNode : ConverterNode(_lword, _lreal);
	_real_to_lreal_ConverterNode : ConverterNode(_real, _lreal);
	_sint_to_lreal_ConverterNode : ConverterNode(_sint, _lreal);
	_tod_to_lreal_ConverterNode : ConverterNode(_tod, _lreal);
	_udint_to_lreal_ConverterNode : ConverterNode(_udint, _lreal);
	_uint_to_lreal_ConverterNode : ConverterNode(_uint, _lreal);
	_ulint_to_lreal_ConverterNode : ConverterNode(_ulint, _lreal);
	_usint_to_lreal_ConverterNode : ConverterNode(_usint, _lreal);
	_word_to_lreal_ConverterNode : ConverterNode(_word, _lreal);
	_string_to_lreal_ConverterNode : ConverterNode(_string, _lreal);
	
	// _to_lword
	_bool_to_lword_ConverterNode : ConverterNode(_bool, _lword);
	_byte_to_lword_ConverterNode : ConverterNode(_byte, _lword);
	_dint_to_lword_ConverterNode : ConverterNode(_dint, _lword);
	_dt_to_lword_ConverterNode : ConverterNode(_dt, _lword);
	_dword_to_lword_ConverterNode : ConverterNode(_dword, _lword);
	_int_to_lword_ConverterNode : ConverterNode(_int, _lword);
	_lint_to_lword_ConverterNode : ConverterNode(_lint, _lword);
	_lreal_to_lword_ConverterNode : ConverterNode(_lreal, _lword);
	_lword_to_lword_ConverterNode : ConverterNode(_lword, _lword);
	_real_to_lword_ConverterNode : ConverterNode(_real, _lword);
	_sint_to_lword_ConverterNode : ConverterNode(_sint, _lword);
	_tod_to_lword_ConverterNode : ConverterNode(_tod, _lword);
	_udint_to_lword_ConverterNode : ConverterNode(_udint, _lword);
	_uint_to_lword_ConverterNode : ConverterNode(_uint, _lword);
	_ulint_to_lword_ConverterNode : ConverterNode(_ulint, _lword);
	_usint_to_lword_ConverterNode : ConverterNode(_usint, _lword);
	_word_to_lword_ConverterNode : ConverterNode(_word, _lword);
	_string_to_lword_ConverterNode : ConverterNode(_string, _lword);

	// _to_real
	_bool_to_real_ConverterNode : ConverterNode(_bool, _real);
	_byte_to_real_ConverterNode : ConverterNode(_byte, _real);
	_dint_to_real_ConverterNode : ConverterNode(_dint, _real);
	_dt_to_real_ConverterNode : ConverterNode(_dt, _real);
	_dword_to_real_ConverterNode : ConverterNode(_dword, _real);
	_int_to_real_ConverterNode : ConverterNode(_int, _real);
	_lint_to_real_ConverterNode : ConverterNode(_lint, _real);
	_lreal_to_real_ConverterNode : ConverterNode(_lreal, _real);
	_lword_to_real_ConverterNode : ConverterNode(_lword, _real);
	_real_to_real_ConverterNode : ConverterNode(_real, _real);
	_sint_to_real_ConverterNode : ConverterNode(_sint, _real);
	_tod_to_real_ConverterNode : ConverterNode(_tod, _real);
	_udint_to_real_ConverterNode : ConverterNode(_udint, _real);
	_uint_to_real_ConverterNode : ConverterNode(_uint, _real);
	_ulint_to_real_ConverterNode : ConverterNode(_ulint, _real);
	_usint_to_real_ConverterNode : ConverterNode(_usint, _real);
	_word_to_real_ConverterNode : ConverterNode(_word, _real);
	_string_to_real_ConverterNode : ConverterNode(_string, _real);
	
	// _to_sint
	_bool_to_sint_ConverterNode : ConverterNode(_bool, _sint);
	_byte_to_sint_ConverterNode : ConverterNode(_byte, _sint);
	_dint_to_sint_ConverterNode : ConverterNode(_dint, _sint);
	_dt_to_sint_ConverterNode : ConverterNode(_dt, _sint);
	_dword_to_sint_ConverterNode : ConverterNode(_dword, _sint);
	_int_to_sint_ConverterNode : ConverterNode(_int, _sint);
	_lint_to_sint_ConverterNode : ConverterNode(_lint, _sint);
	_lreal_to_sint_ConverterNode : ConverterNode(_lreal, _sint);
	_lword_to_sint_ConverterNode : ConverterNode(_lword, _sint);
	_real_to_sint_ConverterNode : ConverterNode(_real, _sint);
	_sint_to_sint_ConverterNode : ConverterNode(_sint, _sint);
	_tod_to_sint_ConverterNode : ConverterNode(_tod, _sint);
	_udint_to_sint_ConverterNode : ConverterNode(_udint, _sint);
	_uint_to_sint_ConverterNode : ConverterNode(_uint, _sint);
	_ulint_to_sint_ConverterNode : ConverterNode(_ulint, _sint);
	_usint_to_sint_ConverterNode : ConverterNode(_usint, _sint);
	_word_to_sint_ConverterNode : ConverterNode(_word, _sint);
	_string_to_sint_ConverterNode : ConverterNode(_string, _sint);

	// _to_tod
	_bool_to_tod_ConverterNode : ConverterNode(_bool, _tod);
	_byte_to_tod_ConverterNode : ConverterNode(_byte, _tod);
	_dint_to_tod_ConverterNode : ConverterNode(_dint, _tod);
	_dt_to_tod_ConverterNode : ConverterNode(_dt, _tod);
	_dword_to_tod_ConverterNode : ConverterNode(_dword, _tod);
	_int_to_tod_ConverterNode : ConverterNode(_int, _tod);
	_lint_to_tod_ConverterNode : ConverterNode(_lint, _tod);
	_lreal_to_tod_ConverterNode : ConverterNode(_lreal, _tod);
	_lword_to_tod_ConverterNode : ConverterNode(_lword, _tod);
	_real_to_tod_ConverterNode : ConverterNode(_real, _tod);
	_sint_to_tod_ConverterNode : ConverterNode(_sint, _tod);
	_tod_to_tod_ConverterNode : ConverterNode(_tod, _tod);
	_udint_to_tod_ConverterNode : ConverterNode(_udint, _tod);
	_uint_to_tod_ConverterNode : ConverterNode(_uint, _tod);
	_ulint_to_tod_ConverterNode : ConverterNode(_ulint, _tod);
	_usint_to_tod_ConverterNode : ConverterNode(_usint, _tod);
	_word_to_tod_ConverterNode : ConverterNode(_word, _tod);
	_string_to_tod_ConverterNode : ConverterNode(_string, _tod);
	
	// _to_udint
	_bool_to_udint_ConverterNode : ConverterNode(_bool, _udint);
	_byte_to_udint_ConverterNode : ConverterNode(_byte, _udint);
	_dint_to_udint_ConverterNode : ConverterNode(_dint, _udint);
	_dt_to_udint_ConverterNode : ConverterNode(_dt, _udint);
	_dword_to_udint_ConverterNode : ConverterNode(_dword, _udint);
	_int_to_udint_ConverterNode : ConverterNode(_int, _udint);
	_lint_to_udint_ConverterNode : ConverterNode(_lint, _udint);
	_lreal_to_udint_ConverterNode : ConverterNode(_lreal, _udint);
	_lword_to_udint_ConverterNode : ConverterNode(_lword, _udint);
	_real_to_udint_ConverterNode : ConverterNode(_real, _udint);
	_sint_to_udint_ConverterNode : ConverterNode(_sint, _udint);
	_tod_to_udint_ConverterNode : ConverterNode(_tod, _udint);
	_udint_to_udint_ConverterNode : ConverterNode(_udint, _udint);
	_uint_to_udint_ConverterNode : ConverterNode(_uint, _udint);
	_ulint_to_udint_ConverterNode : ConverterNode(_ulint, _udint);
	_usint_to_udint_ConverterNode : ConverterNode(_usint, _udint);
	_word_to_udint_ConverterNode : ConverterNode(_word, _udint);
	_string_to_udint_ConverterNode : ConverterNode(_string, _udint);

	// _to_uint
	_bool_to_uint_ConverterNode : ConverterNode(_bool, _uint);
	_byte_to_uint_ConverterNode : ConverterNode(_byte, _uint);
	_dint_to_uint_ConverterNode : ConverterNode(_dint, _uint);
	_dt_to_uint_ConverterNode : ConverterNode(_dt, _uint);
	_dword_to_uint_ConverterNode : ConverterNode(_dword, _uint);
	_int_to_uint_ConverterNode : ConverterNode(_int, _uint);
	_lint_to_uint_ConverterNode : ConverterNode(_lint, _uint);
	_lreal_to_uint_ConverterNode : ConverterNode(_lreal, _uint);
	_lword_to_uint_ConverterNode : ConverterNode(_lword, _uint);
	_real_to_uint_ConverterNode : ConverterNode(_real, _uint);
	_sint_to_uint_ConverterNode : ConverterNode(_sint, _uint);
	_tod_to_uint_ConverterNode : ConverterNode(_tod, _uint);
	_udint_to_uint_ConverterNode : ConverterNode(_udint, _uint);
	_uint_to_uint_ConverterNode : ConverterNode(_uint, _uint);
	_ulint_to_uint_ConverterNode : ConverterNode(_ulint, _uint);
	_usint_to_uint_ConverterNode : ConverterNode(_usint, _uint);
	_word_to_uint_ConverterNode : ConverterNode(_word, _uint);
	_string_to_uint_ConverterNode : ConverterNode(_string, _uint);
	
	// _to_ulint
	_bool_to_ulint_ConverterNode : ConverterNode(_bool, _ulint);
	_byte_to_ulint_ConverterNode : ConverterNode(_byte, _ulint);
	_dint_to_ulint_ConverterNode : ConverterNode(_dint, _ulint);
	_dt_to_ulint_ConverterNode : ConverterNode(_dt, _ulint);
	_dword_to_ulint_ConverterNode : ConverterNode(_dword, _ulint);
	_int_to_ulint_ConverterNode : ConverterNode(_int, _ulint);
	_lint_to_ulint_ConverterNode : ConverterNode(_lint, _ulint);
	_lreal_to_ulint_ConverterNode : ConverterNode(_lreal, _ulint);
	_lword_to_ulint_ConverterNode : ConverterNode(_lword, _ulint);
	_real_to_ulint_ConverterNode : ConverterNode(_real, _ulint);
	_sint_to_ulint_ConverterNode : ConverterNode(_sint, _ulint);
	_tod_to_ulint_ConverterNode : ConverterNode(_tod, _ulint);
	_udint_to_ulint_ConverterNode : ConverterNode(_udint, _ulint);
	_uint_to_ulint_ConverterNode : ConverterNode(_uint, _ulint);
	_ulint_to_ulint_ConverterNode : ConverterNode(_ulint, _ulint);
	_usint_to_ulint_ConverterNode : ConverterNode(_usint, _ulint);
	_word_to_ulint_ConverterNode : ConverterNode(_word, _ulint);
	_string_to_ulint_ConverterNode : ConverterNode(_string, _ulint);

	// _to_usint
	_bool_to_usint_ConverterNode : ConverterNode(_bool, _usint);
	_byte_to_usint_ConverterNode : ConverterNode(_byte, _usint);
	_dint_to_usint_ConverterNode : ConverterNode(_dint, _usint);
	_dt_to_usint_ConverterNode : ConverterNode(_dt, _usint);
	_dword_to_usint_ConverterNode : ConverterNode(_dword, _usint);
	_int_to_usint_ConverterNode : ConverterNode(_int, _usint);
	_lint_to_usint_ConverterNode : ConverterNode(_lint, _usint);
	_lreal_to_usint_ConverterNode : ConverterNode(_lreal, _usint);
	_lword_to_usint_ConverterNode : ConverterNode(_lword, _usint);
	_real_to_usint_ConverterNode : ConverterNode(_real, _usint);
	_sint_to_usint_ConverterNode : ConverterNode(_sint, _usint);
	_tod_to_usint_ConverterNode : ConverterNode(_tod, _usint);
	_udint_to_usint_ConverterNode : ConverterNode(_udint, _usint);
	_uint_to_usint_ConverterNode : ConverterNode(_uint, _usint);
	_ulint_to_usint_ConverterNode : ConverterNode(_ulint, _usint);
	_usint_to_usint_ConverterNode : ConverterNode(_usint, _usint);
	_word_to_usint_ConverterNode : ConverterNode(_word, _usint);
	_string_to_usint_ConverterNode : ConverterNode(_string, _usint);
	
	// _to_word
	_bool_to_word_ConverterNode : ConverterNode(_bool, _word);
	_byte_to_word_ConverterNode : ConverterNode(_byte, _word);
	_dint_to_word_ConverterNode : ConverterNode(_dint, _word);
	_dt_to_word_ConverterNode : ConverterNode(_dt, _word);
	_dword_to_word_ConverterNode : ConverterNode(_dword, _word);
	_int_to_word_ConverterNode : ConverterNode(_int, _word);
	_lint_to_word_ConverterNode : ConverterNode(_lint, _word);
	_lreal_to_word_ConverterNode : ConverterNode(_lreal, _word);
	_lword_to_word_ConverterNode : ConverterNode(_lword, _word);
	_real_to_word_ConverterNode : ConverterNode(_real, _word);
	_sint_to_word_ConverterNode : ConverterNode(_sint, _word);
	_tod_to_word_ConverterNode : ConverterNode(_tod, _word);
	_udint_to_word_ConverterNode : ConverterNode(_udint, _word);
	_uint_to_word_ConverterNode : ConverterNode(_uint, _word);
	_ulint_to_word_ConverterNode : ConverterNode(_ulint, _word);
	_usint_to_word_ConverterNode : ConverterNode(_usint, _word);
	_word_to_word_ConverterNode : ConverterNode(_word, _word);
	_string_to_word_ConverterNode : ConverterNode(_string, _word);

	// _to_string
	_bool_to_string_ConverterNode : ConverterNode(_bool, _string);
	_byte_to_string_ConverterNode : ConverterNode(_byte, _string);
	_dint_to_string_ConverterNode : ConverterNode(_dint, _string);
	_dt_to_string_ConverterNode : ConverterNode(_dt, _string);
	_dword_to_string_ConverterNode : ConverterNode(_dword, _string);
	_int_to_string_ConverterNode : ConverterNode(_int, _string);
	_lint_to_string_ConverterNode : ConverterNode(_lint, _string);
	_lreal_to_string_ConverterNode : ConverterNode(_lreal, _string);
	_lword_to_string_ConverterNode : ConverterNode(_lword, _string);
	_real_to_string_ConverterNode : ConverterNode(_real, _string);
	_sint_to_string_ConverterNode : ConverterNode(_sint, _string);
	_tod_to_string_ConverterNode : ConverterNode(_tod, _string);
	_udint_to_string_ConverterNode : ConverterNode(_udint, _string);
	_uint_to_string_ConverterNode : ConverterNode(_uint, _string);
	_ulint_to_string_ConverterNode : ConverterNode(_ulint, _string);
	_usint_to_string_ConverterNode : ConverterNode(_usint, _string);
	_word_to_string_ConverterNode : ConverterNode(_word, _string);
	_string_to_string_ConverterNode : ConverterNode(_string, _string);
END_VAR

METHOD PUBLIC Register
VAR_INPUT
	Datatypes : I_Datatypes;
	NodeFactory : I_NodeFactory;
END_VAR
Datatypes.RegisterDatatype(_bool);
Datatypes.RegisterDatatype(_byte);
Datatypes.RegisterDatatype(_dint);
Datatypes.RegisterDatatype(_dt);
Datatypes.RegisterDatatype(_dword);
Datatypes.RegisterDatatype(_int);
Datatypes.RegisterDatatype(_lint);
Datatypes.RegisterDatatype(_lreal);
Datatypes.RegisterDatatype(_lword);
Datatypes.RegisterDatatype(_real);
Datatypes.RegisterDatatype(_sint);
Datatypes.RegisterDatatype(_time_of_day);
Datatypes.RegisterDatatype(_tod);
Datatypes.RegisterDatatype(_udint);
Datatypes.RegisterDatatype(_uint);
Datatypes.RegisterDatatype(_ulint);
Datatypes.RegisterDatatype(_usint);
Datatypes.RegisterDatatype(_word);
Datatypes.RegisterDatatype(_string);
Datatypes.RegisterDatatype(_pvoid);

// _to_byte
NodeFactory.AddNodeAsPrototype('IEC Datatypes/Converters/TO_BOOL/BOOL_TO_BOOL', _bool_to_bool_ConverterNode);
NodeFactory.AddNodeAsPrototype('IEC Datatypes/Converters/TO_BOOL/BYTE_TO_BOOL', _byte_to_bool_ConverterNode);
NodeFactory.AddNodeAsPrototype('IEC Datatypes/Converters/TO_BOOL/DINT_TO_BOOL', _dint_to_bool_ConverterNode);
NodeFactory.AddNodeAsPrototype('IEC Datatypes/Converters/TO_BOOL/DT_TO_BOOL', _dt_to_bool_ConverterNode);
NodeFactory.AddNodeAsPrototype('IEC Datatypes/Converters/TO_BOOL/DWORD_TO_BOOL', _dword_to_bool_ConverterNode);
NodeFactory.AddNodeAsPrototype('IEC Datatypes/Converters/TO_BOOL/INT_TO_BOOL', _int_to_bool_ConverterNode);
NodeFactory.AddNodeAsPrototype('IEC Datatypes/Converters/TO_BOOL/LINT_TO_BOOL', _lint_to_bool_ConverterNode);
NodeFactory.AddNodeAsPrototype('IEC Datatypes/Converters/TO_BOOL/LREAL_TO_BOOL', _lreal_to_bool_ConverterNode);
NodeFactory.AddNodeAsPrototype('IEC Datatypes/Converters/TO_BOOL/LWORD_TO_BOOL', _lword_to_bool_ConverterNode);
NodeFactory.AddNodeAsPrototype('IEC Datatypes/Converters/TO_BOOL/REAL_TO_BOOL', _real_to_bool_ConverterNode);
NodeFactory.AddNodeAsPrototype('IEC Datatypes/Converters/TO_BOOL/SINT_TO_BOOL', _sint_to_bool_ConverterNode);
NodeFactory.AddNodeAsPrototype('IEC Datatypes/Converters/TO_BOOL/TOD_TO_BOOL', _tod_to_bool_ConverterNode);
NodeFactory.AddNodeAsPrototype('IEC Datatypes/Converters/TO_BOOL/UDINT_TO_BOOL', _udint_to_bool_ConverterNode);
NodeFactory.AddNodeAsPrototype('IEC Datatypes/Converters/TO_BOOL/UINT_TO_BOOL', _uint_to_bool_ConverterNode);
NodeFactory.AddNodeAsPrototype('IEC Datatypes/Converters/TO_BOOL/ULINT_TO_BOOL', _ulint_to_bool_ConverterNode);
NodeFactory.AddNodeAsPrototype('IEC Datatypes/Converters/TO_BOOL/USINT_TO_BOOL', _usint_to_bool_ConverterNode);
NodeFactory.AddNodeAsPrototype('IEC Datatypes/Converters/TO_BOOL/WORD_TO_BOOL', _word_to_bool_ConverterNode);
NodeFactory.AddNodeAsPrototype('IEC Datatypes/Converters/TO_BOOL/STRING_TO_BOOL', _string_to_bool_ConverterNode);

// _to_byte
NodeFactory.AddNodeAsPrototype('IEC Datatypes/Converters/TO_BYTE/BOOL_TO_BYTE', _bool_to_byte_ConverterNode);
NodeFactory.AddNodeAsPrototype('IEC Datatypes/Converters/TO_BYTE/BYTE_TO_BYTE', _byte_to_byte_ConverterNode);
NodeFactory.AddNodeAsPrototype('IEC Datatypes/Converters/TO_BYTE/DINT_TO_BYTE', _dint_to_byte_ConverterNode);
NodeFactory.AddNodeAsPrototype('IEC Datatypes/Converters/TO_BYTE/DT_TO_BYTE', _dt_to_byte_ConverterNode);
NodeFactory.AddNodeAsPrototype('IEC Datatypes/Converters/TO_BYTE/DWORD_TO_BYTE', _dword_to_byte_ConverterNode);
NodeFactory.AddNodeAsPrototype('IEC Datatypes/Converters/TO_BYTE/INT_TO_BYTE', _int_to_byte_ConverterNode);
NodeFactory.AddNodeAsPrototype('IEC Datatypes/Converters/TO_BYTE/LINT_TO_BYTE', _lint_to_byte_ConverterNode);
NodeFactory.AddNodeAsPrototype('IEC Datatypes/Converters/TO_BYTE/LREAL_TO_BYTE', _lreal_to_byte_ConverterNode);
NodeFactory.AddNodeAsPrototype('IEC Datatypes/Converters/TO_BYTE/LWORD_TO_BYTE', _lword_to_byte_ConverterNode);
NodeFactory.AddNodeAsPrototype('IEC Datatypes/Converters/TO_BYTE/REAL_TO_BYTE', _real_to_byte_ConverterNode);
NodeFactory.AddNodeAsPrototype('IEC Datatypes/Converters/TO_BYTE/SINT_TO_BYTE', _sint_to_byte_ConverterNode);
NodeFactory.AddNodeAsPrototype('IEC Datatypes/Converters/TO_BYTE/TOD_TO_BYTE', _tod_to_byte_ConverterNode);
NodeFactory.AddNodeAsPrototype('IEC Datatypes/Converters/TO_BYTE/UDINT_TO_BYTE', _udint_to_byte_ConverterNode);
NodeFactory.AddNodeAsPrototype('IEC Datatypes/Converters/TO_BYTE/UINT_TO_BYTE', _uint_to_byte_ConverterNode);
NodeFactory.AddNodeAsPrototype('IEC Datatypes/Converters/TO_BYTE/ULINT_TO_BYTE', _ulint_to_byte_ConverterNode);
NodeFactory.AddNodeAsPrototype('IEC Datatypes/Converters/TO_BYTE/USINT_TO_BYTE', _usint_to_byte_ConverterNode);
NodeFactory.AddNodeAsPrototype('IEC Datatypes/Converters/TO_BYTE/WORD_TO_BYTE', _word_to_byte_ConverterNode);
NodeFactory.AddNodeAsPrototype('IEC Datatypes/Converters/TO_BYTE/STRING_TO_BYTE', _string_to_byte_ConverterNode);

// _to_dint
NodeFactory.AddNodeAsPrototype('IEC Datatypes/Converters/TO_DINT/BOOL_TO_DINT', _bool_to_dint_ConverterNode);
NodeFactory.AddNodeAsPrototype('IEC Datatypes/Converters/TO_DINT/BYTE_TO_DINT', _byte_to_dint_ConverterNode);
NodeFactory.AddNodeAsPrototype('IEC Datatypes/Converters/TO_DINT/DINT_TO_DINT', _dint_to_dint_ConverterNode);
NodeFactory.AddNodeAsPrototype('IEC Datatypes/Converters/TO_DINT/DT_TO_DINT', _dt_to_dint_ConverterNode);
NodeFactory.AddNodeAsPrototype('IEC Datatypes/Converters/TO_DINT/DWORD_TO_DINT', _dword_to_dint_ConverterNode);
NodeFactory.AddNodeAsPrototype('IEC Datatypes/Converters/TO_DINT/INT_TO_DINT', _int_to_dint_ConverterNode);
NodeFactory.AddNodeAsPrototype('IEC Datatypes/Converters/TO_DINT/LINT_TO_DINT', _lint_to_dint_ConverterNode);
NodeFactory.AddNodeAsPrototype('IEC Datatypes/Converters/TO_DINT/LREAL_TO_DINT', _lreal_to_dint_ConverterNode);
NodeFactory.AddNodeAsPrototype('IEC Datatypes/Converters/TO_DINT/LWORD_TO_DINT', _lword_to_dint_ConverterNode);
NodeFactory.AddNodeAsPrototype('IEC Datatypes/Converters/TO_DINT/REAL_TO_DINT', _real_to_dint_ConverterNode);
NodeFactory.AddNodeAsPrototype('IEC Datatypes/Converters/TO_DINT/SINT_TO_DINT', _sint_to_dint_ConverterNode);
NodeFactory.AddNodeAsPrototype('IEC Datatypes/Converters/TO_DINT/TOD_TO_DINT', _tod_to_dint_ConverterNode);
NodeFactory.AddNodeAsPrototype('IEC Datatypes/Converters/TO_DINT/UDINT_TO_DINT', _udint_to_dint_ConverterNode);
NodeFactory.AddNodeAsPrototype('IEC Datatypes/Converters/TO_DINT/UINT_TO_DINT', _uint_to_dint_ConverterNode);
NodeFactory.AddNodeAsPrototype('IEC Datatypes/Converters/TO_DINT/ULINT_TO_DINT', _ulint_to_dint_ConverterNode);
NodeFactory.AddNodeAsPrototype('IEC Datatypes/Converters/TO_DINT/USINT_TO_DINT', _usint_to_dint_ConverterNode);
NodeFactory.AddNodeAsPrototype('IEC Datatypes/Converters/TO_DINT/WORD_TO_DINT', _word_to_dint_ConverterNode);
NodeFactory.AddNodeAsPrototype('IEC Datatypes/Converters/TO_DINT/STRING_TO_DINT', _string_to_dint_ConverterNode);

// _to_dt
NodeFactory.AddNodeAsPrototype('IEC Datatypes/Converters/TO_DT/BOOL_TO_DT', _bool_to_dt_ConverterNode);
NodeFactory.AddNodeAsPrototype('IEC Datatypes/Converters/TO_DT/BYTE_TO_DT', _byte_to_dt_ConverterNode);
NodeFactory.AddNodeAsPrototype('IEC Datatypes/Converters/TO_DT/DINT_TO_DT', _dint_to_dt_ConverterNode);
NodeFactory.AddNodeAsPrototype('IEC Datatypes/Converters/TO_DT/DT_TO_DT', _dt_to_dt_ConverterNode);
NodeFactory.AddNodeAsPrototype('IEC Datatypes/Converters/TO_DT/DWORD_TO_DT', _dword_to_dt_ConverterNode);
NodeFactory.AddNodeAsPrototype('IEC Datatypes/Converters/TO_DT/INT_TO_DT', _int_to_dt_ConverterNode);
NodeFactory.AddNodeAsPrototype('IEC Datatypes/Converters/TO_DT/LINT_TO_DT', _lint_to_dt_ConverterNode);
NodeFactory.AddNodeAsPrototype('IEC Datatypes/Converters/TO_DT/LREAL_TO_DT', _lreal_to_dt_ConverterNode);
NodeFactory.AddNodeAsPrototype('IEC Datatypes/Converters/TO_DT/LWORD_TO_DT', _lword_to_dt_ConverterNode);
NodeFactory.AddNodeAsPrototype('IEC Datatypes/Converters/TO_DT/REAL_TO_DT', _real_to_dt_ConverterNode);
NodeFactory.AddNodeAsPrototype('IEC Datatypes/Converters/TO_DT/SINT_TO_DT', _sint_to_dt_ConverterNode);
NodeFactory.AddNodeAsPrototype('IEC Datatypes/Converters/TO_DT/TOD_TO_DT', _tod_to_dt_ConverterNode);
NodeFactory.AddNodeAsPrototype('IEC Datatypes/Converters/TO_DT/UDINT_TO_DT', _udint_to_dt_ConverterNode);
NodeFactory.AddNodeAsPrototype('IEC Datatypes/Converters/TO_DT/UINT_TO_DT', _uint_to_dt_ConverterNode);
NodeFactory.AddNodeAsPrototype('IEC Datatypes/Converters/TO_DT/ULINT_TO_DT', _ulint_to_dt_ConverterNode);
NodeFactory.AddNodeAsPrototype('IEC Datatypes/Converters/TO_DT/USINT_TO_DT', _usint_to_dt_ConverterNode);
NodeFactory.AddNodeAsPrototype('IEC Datatypes/Converters/TO_DT/WORD_TO_DT', _word_to_dt_ConverterNode);
NodeFactory.AddNodeAsPrototype('IEC Datatypes/Converters/TO_DT/STRING_TO_DT', _string_to_dt_ConverterNode);

// _to_dword
NodeFactory.AddNodeAsPrototype('IEC Datatypes/Converters/TO_DWORD/BOOL_TO_DWORD', _bool_to_dword_ConverterNode);
NodeFactory.AddNodeAsPrototype('IEC Datatypes/Converters/TO_DWORD/BYTE_TO_DWORD', _byte_to_dword_ConverterNode);
NodeFactory.AddNodeAsPrototype('IEC Datatypes/Converters/TO_DWORD/DINT_TO_DWORD', _dint_to_dword_ConverterNode);
NodeFactory.AddNodeAsPrototype('IEC Datatypes/Converters/TO_DWORD/DT_TO_DWORD', _dt_to_dword_ConverterNode);
NodeFactory.AddNodeAsPrototype('IEC Datatypes/Converters/TO_DWORD/DWORD_TO_DWORD', _dword_to_dword_ConverterNode);
NodeFactory.AddNodeAsPrototype('IEC Datatypes/Converters/TO_DWORD/INT_TO_DWORD', _int_to_dword_ConverterNode);
NodeFactory.AddNodeAsPrototype('IEC Datatypes/Converters/TO_DWORD/LINT_TO_DWORD', _lint_to_dword_ConverterNode);
NodeFactory.AddNodeAsPrototype('IEC Datatypes/Converters/TO_DWORD/LREAL_TO_DWORD', _lreal_to_dword_ConverterNode);
NodeFactory.AddNodeAsPrototype('IEC Datatypes/Converters/TO_DWORD/LWORD_TO_DWORD', _lword_to_dword_ConverterNode);
NodeFactory.AddNodeAsPrototype('IEC Datatypes/Converters/TO_DWORD/REAL_TO_DWORD', _real_to_dword_ConverterNode);
NodeFactory.AddNodeAsPrototype('IEC Datatypes/Converters/TO_DWORD/SINT_TO_DWORD', _sint_to_dword_ConverterNode);
NodeFactory.AddNodeAsPrototype('IEC Datatypes/Converters/TO_DWORD/TOD_TO_DWORD', _tod_to_dword_ConverterNode);
NodeFactory.AddNodeAsPrototype('IEC Datatypes/Converters/TO_DWORD/UDINT_TO_DWORD', _udint_to_dword_ConverterNode);
NodeFactory.AddNodeAsPrototype('IEC Datatypes/Converters/TO_DWORD/UINT_TO_DWORD', _uint_to_dword_ConverterNode);
NodeFactory.AddNodeAsPrototype('IEC Datatypes/Converters/TO_DWORD/ULINT_TO_DWORD', _ulint_to_dword_ConverterNode);
NodeFactory.AddNodeAsPrototype('IEC Datatypes/Converters/TO_DWORD/USINT_TO_DWORD', _usint_to_dword_ConverterNode);
NodeFactory.AddNodeAsPrototype('IEC Datatypes/Converters/TO_DWORD/WORD_TO_DWORD', _word_to_dword_ConverterNode);
NodeFactory.AddNodeAsPrototype('IEC Datatypes/Converters/TO_DWORD/STRING_TO_DWORD', _string_to_dword_ConverterNode);

// _to_int
NodeFactory.AddNodeAsPrototype('IEC Datatypes/Converters/TO_INT/BOOL_TO_INT', _bool_to_int_ConverterNode);
NodeFactory.AddNodeAsPrototype('IEC Datatypes/Converters/TO_INT/BYTE_TO_INT', _byte_to_int_ConverterNode);
NodeFactory.AddNodeAsPrototype('IEC Datatypes/Converters/TO_INT/DINT_TO_INT', _dint_to_int_ConverterNode);
NodeFactory.AddNodeAsPrototype('IEC Datatypes/Converters/TO_INT/DT_TO_INT', _dt_to_int_ConverterNode);
NodeFactory.AddNodeAsPrototype('IEC Datatypes/Converters/TO_INT/DWORD_TO_INT', _dword_to_int_ConverterNode);
NodeFactory.AddNodeAsPrototype('IEC Datatypes/Converters/TO_INT/INT_TO_INT', _int_to_int_ConverterNode);
NodeFactory.AddNodeAsPrototype('IEC Datatypes/Converters/TO_INT/LINT_TO_INT', _lint_to_int_ConverterNode);
NodeFactory.AddNodeAsPrototype('IEC Datatypes/Converters/TO_INT/LREAL_TO_INT', _lreal_to_int_ConverterNode);
NodeFactory.AddNodeAsPrototype('IEC Datatypes/Converters/TO_INT/LWORD_TO_INT', _lword_to_int_ConverterNode);
NodeFactory.AddNodeAsPrototype('IEC Datatypes/Converters/TO_INT/REAL_TO_INT', _real_to_int_ConverterNode);
NodeFactory.AddNodeAsPrototype('IEC Datatypes/Converters/TO_INT/SINT_TO_INT', _sint_to_int_ConverterNode);
NodeFactory.AddNodeAsPrototype('IEC Datatypes/Converters/TO_INT/TOD_TO_INT', _tod_to_int_ConverterNode);
NodeFactory.AddNodeAsPrototype('IEC Datatypes/Converters/TO_INT/UDINT_TO_INT', _udint_to_int_ConverterNode);
NodeFactory.AddNodeAsPrototype('IEC Datatypes/Converters/TO_INT/UINT_TO_INT', _uint_to_int_ConverterNode);
NodeFactory.AddNodeAsPrototype('IEC Datatypes/Converters/TO_INT/ULINT_TO_INT', _ulint_to_int_ConverterNode);
NodeFactory.AddNodeAsPrototype('IEC Datatypes/Converters/TO_INT/USINT_TO_INT', _usint_to_int_ConverterNode);
NodeFactory.AddNodeAsPrototype('IEC Datatypes/Converters/TO_INT/WORD_TO_INT', _word_to_int_ConverterNode);
NodeFactory.AddNodeAsPrototype('IEC Datatypes/Converters/TO_INT/STRING_TO_INT', _string_to_int_ConverterNode);

// _to_lint
NodeFactory.AddNodeAsPrototype('IEC Datatypes/Converters/TO_LINT/BOOL_TO_LINT', _bool_to_lint_ConverterNode);
NodeFactory.AddNodeAsPrototype('IEC Datatypes/Converters/TO_LINT/BYTE_TO_LINT', _byte_to_lint_ConverterNode);
NodeFactory.AddNodeAsPrototype('IEC Datatypes/Converters/TO_LINT/DINT_TO_LINT', _dint_to_lint_ConverterNode);
NodeFactory.AddNodeAsPrototype('IEC Datatypes/Converters/TO_LINT/DT_TO_LINT', _dt_to_lint_ConverterNode);
NodeFactory.AddNodeAsPrototype('IEC Datatypes/Converters/TO_LINT/DWORD_TO_LINT', _dword_to_lint_ConverterNode);
NodeFactory.AddNodeAsPrototype('IEC Datatypes/Converters/TO_LINT/INT_TO_LINT', _int_to_lint_ConverterNode);
NodeFactory.AddNodeAsPrototype('IEC Datatypes/Converters/TO_LINT/LINT_TO_LINT', _lint_to_lint_ConverterNode);
NodeFactory.AddNodeAsPrototype('IEC Datatypes/Converters/TO_LINT/LREAL_TO_LINT', _lreal_to_lint_ConverterNode);
NodeFactory.AddNodeAsPrototype('IEC Datatypes/Converters/TO_LINT/LWORD_TO_LINT', _lword_to_lint_ConverterNode);
NodeFactory.AddNodeAsPrototype('IEC Datatypes/Converters/TO_LINT/REAL_TO_LINT', _real_to_lint_ConverterNode);
NodeFactory.AddNodeAsPrototype('IEC Datatypes/Converters/TO_LINT/SINT_TO_LINT', _sint_to_lint_ConverterNode);
NodeFactory.AddNodeAsPrototype('IEC Datatypes/Converters/TO_LINT/TOD_TO_LINT', _tod_to_lint_ConverterNode);
NodeFactory.AddNodeAsPrototype('IEC Datatypes/Converters/TO_LINT/UDINT_TO_LINT', _udint_to_lint_ConverterNode);
NodeFactory.AddNodeAsPrototype('IEC Datatypes/Converters/TO_LINT/UINT_TO_LINT', _uint_to_lint_ConverterNode);
NodeFactory.AddNodeAsPrototype('IEC Datatypes/Converters/TO_LINT/ULINT_TO_LINT', _ulint_to_lint_ConverterNode);
NodeFactory.AddNodeAsPrototype('IEC Datatypes/Converters/TO_LINT/USINT_TO_LINT', _usint_to_lint_ConverterNode);
NodeFactory.AddNodeAsPrototype('IEC Datatypes/Converters/TO_LINT/WORD_TO_LINT', _word_to_lint_ConverterNode);
NodeFactory.AddNodeAsPrototype('IEC Datatypes/Converters/TO_LINT/STRING_TO_LINT', _string_to_lint_ConverterNode);

// _to_lreal
NodeFactory.AddNodeAsPrototype('IEC Datatypes/Converters/TO_LREAL/BOOL_TO_LREAL', _bool_to_lreal_ConverterNode);
NodeFactory.AddNodeAsPrototype('IEC Datatypes/Converters/TO_LREAL/BYTE_TO_LREAL', _byte_to_lreal_ConverterNode);
NodeFactory.AddNodeAsPrototype('IEC Datatypes/Converters/TO_LREAL/DINT_TO_LREAL', _dint_to_lreal_ConverterNode);
NodeFactory.AddNodeAsPrototype('IEC Datatypes/Converters/TO_LREAL/DT_TO_LREAL', _dt_to_lreal_ConverterNode);
NodeFactory.AddNodeAsPrototype('IEC Datatypes/Converters/TO_LREAL/DWORD_TO_LREAL', _dword_to_lreal_ConverterNode);
NodeFactory.AddNodeAsPrototype('IEC Datatypes/Converters/TO_LREAL/INT_TO_LREAL', _int_to_lreal_ConverterNode);
NodeFactory.AddNodeAsPrototype('IEC Datatypes/Converters/TO_LREAL/LINT_TO_LREAL', _lint_to_lreal_ConverterNode);
NodeFactory.AddNodeAsPrototype('IEC Datatypes/Converters/TO_LREAL/LREAL_TO_LREAL', _lreal_to_lreal_ConverterNode);
NodeFactory.AddNodeAsPrototype('IEC Datatypes/Converters/TO_LREAL/LWORD_TO_LREAL', _lword_to_lreal_ConverterNode);
NodeFactory.AddNodeAsPrototype('IEC Datatypes/Converters/TO_LREAL/REAL_TO_LREAL', _real_to_lreal_ConverterNode);
NodeFactory.AddNodeAsPrototype('IEC Datatypes/Converters/TO_LREAL/SINT_TO_LREAL', _sint_to_lreal_ConverterNode);
NodeFactory.AddNodeAsPrototype('IEC Datatypes/Converters/TO_LREAL/TOD_TO_LREAL', _tod_to_lreal_ConverterNode);
NodeFactory.AddNodeAsPrototype('IEC Datatypes/Converters/TO_LREAL/UDINT_TO_LREAL', _udint_to_lreal_ConverterNode);
NodeFactory.AddNodeAsPrototype('IEC Datatypes/Converters/TO_LREAL/UINT_TO_LREAL', _uint_to_lreal_ConverterNode);
NodeFactory.AddNodeAsPrototype('IEC Datatypes/Converters/TO_LREAL/ULINT_TO_LREAL', _ulint_to_lreal_ConverterNode);
NodeFactory.AddNodeAsPrototype('IEC Datatypes/Converters/TO_LREAL/USINT_TO_LREAL', _usint_to_lreal_ConverterNode);
NodeFactory.AddNodeAsPrototype('IEC Datatypes/Converters/TO_LREAL/WORD_TO_LREAL', _word_to_lreal_ConverterNode);
NodeFactory.AddNodeAsPrototype('IEC Datatypes/Converters/TO_LREAL/STRING_TO_LREAL', _string_to_lreal_ConverterNode);

// _to_lword
NodeFactory.AddNodeAsPrototype('IEC Datatypes/Converters/TO_LWORD/BOOL_TO_LWORD', _bool_to_lword_ConverterNode);
NodeFactory.AddNodeAsPrototype('IEC Datatypes/Converters/TO_LWORD/BYTE_TO_LWORD', _byte_to_lword_ConverterNode);
NodeFactory.AddNodeAsPrototype('IEC Datatypes/Converters/TO_LWORD/DINT_TO_LWORD', _dint_to_lword_ConverterNode);
NodeFactory.AddNodeAsPrototype('IEC Datatypes/Converters/TO_LWORD/DT_TO_LWORD', _dt_to_lword_ConverterNode);
NodeFactory.AddNodeAsPrototype('IEC Datatypes/Converters/TO_LWORD/DWORD_TO_LWORD', _dword_to_lword_ConverterNode);
NodeFactory.AddNodeAsPrototype('IEC Datatypes/Converters/TO_LWORD/INT_TO_LWORD', _int_to_lword_ConverterNode);
NodeFactory.AddNodeAsPrototype('IEC Datatypes/Converters/TO_LWORD/LINT_TO_LWORD', _lint_to_lword_ConverterNode);
NodeFactory.AddNodeAsPrototype('IEC Datatypes/Converters/TO_LWORD/LREAL_TO_LWORD', _lreal_to_lword_ConverterNode);
NodeFactory.AddNodeAsPrototype('IEC Datatypes/Converters/TO_LWORD/LWORD_TO_LWORD', _lword_to_lword_ConverterNode);
NodeFactory.AddNodeAsPrototype('IEC Datatypes/Converters/TO_LWORD/REAL_TO_LWORD', _real_to_lword_ConverterNode);
NodeFactory.AddNodeAsPrototype('IEC Datatypes/Converters/TO_LWORD/SINT_TO_LWORD', _sint_to_lword_ConverterNode);
NodeFactory.AddNodeAsPrototype('IEC Datatypes/Converters/TO_LWORD/TOD_TO_LWORD', _tod_to_lword_ConverterNode);
NodeFactory.AddNodeAsPrototype('IEC Datatypes/Converters/TO_LWORD/UDINT_TO_LWORD', _udint_to_lword_ConverterNode);
NodeFactory.AddNodeAsPrototype('IEC Datatypes/Converters/TO_LWORD/UINT_TO_LWORD', _uint_to_lword_ConverterNode);
NodeFactory.AddNodeAsPrototype('IEC Datatypes/Converters/TO_LWORD/ULINT_TO_LWORD', _ulint_to_lword_ConverterNode);
NodeFactory.AddNodeAsPrototype('IEC Datatypes/Converters/TO_LWORD/USINT_TO_LWORD', _usint_to_lword_ConverterNode);
NodeFactory.AddNodeAsPrototype('IEC Datatypes/Converters/TO_LWORD/WORD_TO_LWORD', _word_to_lword_ConverterNode);
NodeFactory.AddNodeAsPrototype('IEC Datatypes/Converters/TO_LWORD/STRING_TO_LWORD', _string_to_lword_ConverterNode);

// _to_real
NodeFactory.AddNodeAsPrototype('IEC Datatypes/Converters/TO_REAL/BOOL_TO_REAL', _bool_to_real_ConverterNode);
NodeFactory.AddNodeAsPrototype('IEC Datatypes/Converters/TO_REAL/BYTE_TO_REAL', _byte_to_real_ConverterNode);
NodeFactory.AddNodeAsPrototype('IEC Datatypes/Converters/TO_REAL/DINT_TO_REAL', _dint_to_real_ConverterNode);
NodeFactory.AddNodeAsPrototype('IEC Datatypes/Converters/TO_REAL/DT_TO_REAL', _dt_to_real_ConverterNode);
NodeFactory.AddNodeAsPrototype('IEC Datatypes/Converters/TO_REAL/DWORD_TO_REAL', _dword_to_real_ConverterNode);
NodeFactory.AddNodeAsPrototype('IEC Datatypes/Converters/TO_REAL/INT_TO_REAL', _int_to_real_ConverterNode);
NodeFactory.AddNodeAsPrototype('IEC Datatypes/Converters/TO_REAL/LINT_TO_REAL', _lint_to_real_ConverterNode);
NodeFactory.AddNodeAsPrototype('IEC Datatypes/Converters/TO_REAL/LREAL_TO_REAL', _lreal_to_real_ConverterNode);
NodeFactory.AddNodeAsPrototype('IEC Datatypes/Converters/TO_REAL/LWORD_TO_REAL', _lword_to_real_ConverterNode);
NodeFactory.AddNodeAsPrototype('IEC Datatypes/Converters/TO_REAL/REAL_TO_REAL', _real_to_real_ConverterNode);
NodeFactory.AddNodeAsPrototype('IEC Datatypes/Converters/TO_REAL/SINT_TO_REAL', _sint_to_real_ConverterNode);
NodeFactory.AddNodeAsPrototype('IEC Datatypes/Converters/TO_REAL/TOD_TO_REAL', _tod_to_real_ConverterNode);
NodeFactory.AddNodeAsPrototype('IEC Datatypes/Converters/TO_REAL/UDINT_TO_REAL', _udint_to_real_ConverterNode);
NodeFactory.AddNodeAsPrototype('IEC Datatypes/Converters/TO_REAL/UINT_TO_REAL', _uint_to_real_ConverterNode);
NodeFactory.AddNodeAsPrototype('IEC Datatypes/Converters/TO_REAL/ULINT_TO_REAL', _ulint_to_real_ConverterNode);
NodeFactory.AddNodeAsPrototype('IEC Datatypes/Converters/TO_REAL/USINT_TO_REAL', _usint_to_real_ConverterNode);
NodeFactory.AddNodeAsPrototype('IEC Datatypes/Converters/TO_REAL/WORD_TO_REAL', _word_to_real_ConverterNode);
NodeFactory.AddNodeAsPrototype('IEC Datatypes/Converters/TO_REAL/STRING_TO_REAL', _string_to_real_ConverterNode);

// _to_sint
NodeFactory.AddNodeAsPrototype('IEC Datatypes/Converters/TO_SINT/BOOL_TO_SINT', _bool_to_sint_ConverterNode);
NodeFactory.AddNodeAsPrototype('IEC Datatypes/Converters/TO_SINT/BYTE_TO_SINT', _byte_to_sint_ConverterNode);
NodeFactory.AddNodeAsPrototype('IEC Datatypes/Converters/TO_SINT/DINT_TO_SINT', _dint_to_sint_ConverterNode);
NodeFactory.AddNodeAsPrototype('IEC Datatypes/Converters/TO_SINT/DT_TO_SINT', _dt_to_sint_ConverterNode);
NodeFactory.AddNodeAsPrototype('IEC Datatypes/Converters/TO_SINT/DWORD_TO_SINT', _dword_to_sint_ConverterNode);
NodeFactory.AddNodeAsPrototype('IEC Datatypes/Converters/TO_SINT/INT_TO_SINT', _int_to_sint_ConverterNode);
NodeFactory.AddNodeAsPrototype('IEC Datatypes/Converters/TO_SINT/LINT_TO_SINT', _lint_to_sint_ConverterNode);
NodeFactory.AddNodeAsPrototype('IEC Datatypes/Converters/TO_SINT/LREAL_TO_SINT', _lreal_to_sint_ConverterNode);
NodeFactory.AddNodeAsPrototype('IEC Datatypes/Converters/TO_SINT/LWORD_TO_SINT', _lword_to_sint_ConverterNode);
NodeFactory.AddNodeAsPrototype('IEC Datatypes/Converters/TO_SINT/REAL_TO_SINT', _real_to_sint_ConverterNode);
NodeFactory.AddNodeAsPrototype('IEC Datatypes/Converters/TO_SINT/SINT_TO_SINT', _sint_to_sint_ConverterNode);
NodeFactory.AddNodeAsPrototype('IEC Datatypes/Converters/TO_SINT/TOD_TO_SINT', _tod_to_sint_ConverterNode);
NodeFactory.AddNodeAsPrototype('IEC Datatypes/Converters/TO_SINT/UDINT_TO_SINT', _udint_to_sint_ConverterNode);
NodeFactory.AddNodeAsPrototype('IEC Datatypes/Converters/TO_SINT/UINT_TO_SINT', _uint_to_sint_ConverterNode);
NodeFactory.AddNodeAsPrototype('IEC Datatypes/Converters/TO_SINT/ULINT_TO_SINT', _ulint_to_sint_ConverterNode);
NodeFactory.AddNodeAsPrototype('IEC Datatypes/Converters/TO_SINT/USINT_TO_SINT', _usint_to_sint_ConverterNode);
NodeFactory.AddNodeAsPrototype('IEC Datatypes/Converters/TO_SINT/WORD_TO_SINT', _word_to_sint_ConverterNode);
NodeFactory.AddNodeAsPrototype('IEC Datatypes/Converters/TO_SINT/STRING_TO_SINT', _string_to_sint_ConverterNode);

// _to_tod
NodeFactory.AddNodeAsPrototype('IEC Datatypes/Converters/TO_TOD/BOOL_TO_TOD', _bool_to_tod_ConverterNode);
NodeFactory.AddNodeAsPrototype('IEC Datatypes/Converters/TO_TOD/BYTE_TO_TOD', _byte_to_tod_ConverterNode);
NodeFactory.AddNodeAsPrototype('IEC Datatypes/Converters/TO_TOD/DINT_TO_TOD', _dint_to_tod_ConverterNode);
NodeFactory.AddNodeAsPrototype('IEC Datatypes/Converters/TO_TOD/DT_TO_TOD', _dt_to_tod_ConverterNode);
NodeFactory.AddNodeAsPrototype('IEC Datatypes/Converters/TO_TOD/DWORD_TO_TOD', _dword_to_tod_ConverterNode);
NodeFactory.AddNodeAsPrototype('IEC Datatypes/Converters/TO_TOD/INT_TO_TOD', _int_to_tod_ConverterNode);
NodeFactory.AddNodeAsPrototype('IEC Datatypes/Converters/TO_TOD/LINT_TO_TOD', _lint_to_tod_ConverterNode);
NodeFactory.AddNodeAsPrototype('IEC Datatypes/Converters/TO_TOD/LREAL_TO_TOD', _lreal_to_tod_ConverterNode);
NodeFactory.AddNodeAsPrototype('IEC Datatypes/Converters/TO_TOD/LWORD_TO_TOD', _lword_to_tod_ConverterNode);
NodeFactory.AddNodeAsPrototype('IEC Datatypes/Converters/TO_TOD/REAL_TO_TOD', _real_to_tod_ConverterNode);
NodeFactory.AddNodeAsPrototype('IEC Datatypes/Converters/TO_TOD/SINT_TO_TOD', _sint_to_tod_ConverterNode);
NodeFactory.AddNodeAsPrototype('IEC Datatypes/Converters/TO_TOD/TOD_TO_TOD', _tod_to_tod_ConverterNode);
NodeFactory.AddNodeAsPrototype('IEC Datatypes/Converters/TO_TOD/UDINT_TO_TOD', _udint_to_tod_ConverterNode);
NodeFactory.AddNodeAsPrototype('IEC Datatypes/Converters/TO_TOD/UINT_TO_TOD', _uint_to_tod_ConverterNode);
NodeFactory.AddNodeAsPrototype('IEC Datatypes/Converters/TO_TOD/ULINT_TO_TOD', _ulint_to_tod_ConverterNode);
NodeFactory.AddNodeAsPrototype('IEC Datatypes/Converters/TO_TOD/USINT_TO_TOD', _usint_to_tod_ConverterNode);
NodeFactory.AddNodeAsPrototype('IEC Datatypes/Converters/TO_TOD/WORD_TO_TOD', _word_to_tod_ConverterNode);
NodeFactory.AddNodeAsPrototype('IEC Datatypes/Converters/TO_TOD/STRING_TO_TOD', _string_to_tod_ConverterNode);

// _to_udint
NodeFactory.AddNodeAsPrototype('IEC Datatypes/Converters/TO_UDINT/BOOL_TO_UDINT', _bool_to_udint_ConverterNode);
NodeFactory.AddNodeAsPrototype('IEC Datatypes/Converters/TO_UDINT/BYTE_TO_UDINT', _byte_to_udint_ConverterNode);
NodeFactory.AddNodeAsPrototype('IEC Datatypes/Converters/TO_UDINT/DINT_TO_UDINT', _dint_to_udint_ConverterNode);
NodeFactory.AddNodeAsPrototype('IEC Datatypes/Converters/TO_UDINT/DT_TO_UDINT', _dt_to_udint_ConverterNode);
NodeFactory.AddNodeAsPrototype('IEC Datatypes/Converters/TO_UDINT/DWORD_TO_UDINT', _dword_to_udint_ConverterNode);
NodeFactory.AddNodeAsPrototype('IEC Datatypes/Converters/TO_UDINT/INT_TO_UDINT', _int_to_udint_ConverterNode);
NodeFactory.AddNodeAsPrototype('IEC Datatypes/Converters/TO_UDINT/LINT_TO_UDINT', _lint_to_udint_ConverterNode);
NodeFactory.AddNodeAsPrototype('IEC Datatypes/Converters/TO_UDINT/LREAL_TO_UDINT', _lreal_to_udint_ConverterNode);
NodeFactory.AddNodeAsPrototype('IEC Datatypes/Converters/TO_UDINT/LWORD_TO_UDINT', _lword_to_udint_ConverterNode);
NodeFactory.AddNodeAsPrototype('IEC Datatypes/Converters/TO_UDINT/REAL_TO_UDINT', _real_to_udint_ConverterNode);
NodeFactory.AddNodeAsPrototype('IEC Datatypes/Converters/TO_UDINT/SINT_TO_UDINT', _sint_to_udint_ConverterNode);
NodeFactory.AddNodeAsPrototype('IEC Datatypes/Converters/TO_UDINT/TOD_TO_UDINT', _tod_to_udint_ConverterNode);
NodeFactory.AddNodeAsPrototype('IEC Datatypes/Converters/TO_UDINT/UDINT_TO_UDINT', _udint_to_udint_ConverterNode);
NodeFactory.AddNodeAsPrototype('IEC Datatypes/Converters/TO_UDINT/UINT_TO_UDINT', _uint_to_udint_ConverterNode);
NodeFactory.AddNodeAsPrototype('IEC Datatypes/Converters/TO_UDINT/ULINT_TO_UDINT', _ulint_to_udint_ConverterNode);
NodeFactory.AddNodeAsPrototype('IEC Datatypes/Converters/TO_UDINT/USINT_TO_UDINT', _usint_to_udint_ConverterNode);
NodeFactory.AddNodeAsPrototype('IEC Datatypes/Converters/TO_UDINT/WORD_TO_UDINT', _word_to_udint_ConverterNode);
NodeFactory.AddNodeAsPrototype('IEC Datatypes/Converters/TO_UDINT/STRING_TO_UDINT', _string_to_udint_ConverterNode);

// _to_uint
NodeFactory.AddNodeAsPrototype('IEC Datatypes/Converters/TO_UINT/BOOL_TO_UINT', _bool_to_uint_ConverterNode);
NodeFactory.AddNodeAsPrototype('IEC Datatypes/Converters/TO_UINT/BYTE_TO_UINT', _byte_to_uint_ConverterNode);
NodeFactory.AddNodeAsPrototype('IEC Datatypes/Converters/TO_UINT/DINT_TO_UINT', _dint_to_uint_ConverterNode);
NodeFactory.AddNodeAsPrototype('IEC Datatypes/Converters/TO_UINT/DT_TO_UINT', _dt_to_uint_ConverterNode);
NodeFactory.AddNodeAsPrototype('IEC Datatypes/Converters/TO_UINT/DWORD_TO_UINT', _dword_to_uint_ConverterNode);
NodeFactory.AddNodeAsPrototype('IEC Datatypes/Converters/TO_UINT/INT_TO_UINT', _int_to_uint_ConverterNode);
NodeFactory.AddNodeAsPrototype('IEC Datatypes/Converters/TO_UINT/LINT_TO_UINT', _lint_to_uint_ConverterNode);
NodeFactory.AddNodeAsPrototype('IEC Datatypes/Converters/TO_UINT/LREAL_TO_UINT', _lreal_to_uint_ConverterNode);
NodeFactory.AddNodeAsPrototype('IEC Datatypes/Converters/TO_UINT/LWORD_TO_UINT', _lword_to_uint_ConverterNode);
NodeFactory.AddNodeAsPrototype('IEC Datatypes/Converters/TO_UINT/REAL_TO_UINT', _real_to_uint_ConverterNode);
NodeFactory.AddNodeAsPrototype('IEC Datatypes/Converters/TO_UINT/SINT_TO_UINT', _sint_to_uint_ConverterNode);
NodeFactory.AddNodeAsPrototype('IEC Datatypes/Converters/TO_UINT/TOD_TO_UINT', _tod_to_uint_ConverterNode);
NodeFactory.AddNodeAsPrototype('IEC Datatypes/Converters/TO_UINT/UDINT_TO_UINT', _udint_to_uint_ConverterNode);
NodeFactory.AddNodeAsPrototype('IEC Datatypes/Converters/TO_UINT/UINT_TO_UINT', _uint_to_uint_ConverterNode);
NodeFactory.AddNodeAsPrototype('IEC Datatypes/Converters/TO_UINT/ULINT_TO_UINT', _ulint_to_uint_ConverterNode);
NodeFactory.AddNodeAsPrototype('IEC Datatypes/Converters/TO_UINT/USINT_TO_UINT', _usint_to_uint_ConverterNode);
NodeFactory.AddNodeAsPrototype('IEC Datatypes/Converters/TO_UINT/WORD_TO_UINT', _word_to_uint_ConverterNode);
NodeFactory.AddNodeAsPrototype('IEC Datatypes/Converters/TO_UINT/STRING_TO_UINT', _string_to_uint_ConverterNode);

// _to_ulint
NodeFactory.AddNodeAsPrototype('IEC Datatypes/Converters/TO_ULINT/BOOL_TO_ULINT', _bool_to_ulint_ConverterNode);
NodeFactory.AddNodeAsPrototype('IEC Datatypes/Converters/TO_ULINT/BYTE_TO_ULINT', _byte_to_ulint_ConverterNode);
NodeFactory.AddNodeAsPrototype('IEC Datatypes/Converters/TO_ULINT/DINT_TO_ULINT', _dint_to_ulint_ConverterNode);
NodeFactory.AddNodeAsPrototype('IEC Datatypes/Converters/TO_ULINT/DT_TO_ULINT', _dt_to_ulint_ConverterNode);
NodeFactory.AddNodeAsPrototype('IEC Datatypes/Converters/TO_ULINT/DWORD_TO_ULINT', _dword_to_ulint_ConverterNode);
NodeFactory.AddNodeAsPrototype('IEC Datatypes/Converters/TO_ULINT/INT_TO_ULINT', _int_to_ulint_ConverterNode);
NodeFactory.AddNodeAsPrototype('IEC Datatypes/Converters/TO_ULINT/LINT_TO_ULINT', _lint_to_ulint_ConverterNode);
NodeFactory.AddNodeAsPrototype('IEC Datatypes/Converters/TO_ULINT/LREAL_TO_ULINT', _lreal_to_ulint_ConverterNode);
NodeFactory.AddNodeAsPrototype('IEC Datatypes/Converters/TO_ULINT/LWORD_TO_ULINT', _lword_to_ulint_ConverterNode);
NodeFactory.AddNodeAsPrototype('IEC Datatypes/Converters/TO_ULINT/REAL_TO_ULINT', _real_to_ulint_ConverterNode);
NodeFactory.AddNodeAsPrototype('IEC Datatypes/Converters/TO_ULINT/SINT_TO_ULINT', _sint_to_ulint_ConverterNode);
NodeFactory.AddNodeAsPrototype('IEC Datatypes/Converters/TO_ULINT/TOD_TO_ULINT', _tod_to_ulint_ConverterNode);
NodeFactory.AddNodeAsPrototype('IEC Datatypes/Converters/TO_ULINT/UDINT_TO_ULINT', _udint_to_ulint_ConverterNode);
NodeFactory.AddNodeAsPrototype('IEC Datatypes/Converters/TO_ULINT/UINT_TO_ULINT', _uint_to_ulint_ConverterNode);
NodeFactory.AddNodeAsPrototype('IEC Datatypes/Converters/TO_ULINT/ULINT_TO_ULINT', _ulint_to_ulint_ConverterNode);
NodeFactory.AddNodeAsPrototype('IEC Datatypes/Converters/TO_ULINT/USINT_TO_ULINT', _usint_to_ulint_ConverterNode);
NodeFactory.AddNodeAsPrototype('IEC Datatypes/Converters/TO_ULINT/WORD_TO_ULINT', _word_to_ulint_ConverterNode);
NodeFactory.AddNodeAsPrototype('IEC Datatypes/Converters/TO_ULINT/STRING_TO_ULINT', _string_to_ulint_ConverterNode);

// _to_usint
NodeFactory.AddNodeAsPrototype('IEC Datatypes/Converters/TO_USINT/BOOL_TO_USINT', _bool_to_usint_ConverterNode);
NodeFactory.AddNodeAsPrototype('IEC Datatypes/Converters/TO_USINT/BYTE_TO_USINT', _byte_to_usint_ConverterNode);
NodeFactory.AddNodeAsPrototype('IEC Datatypes/Converters/TO_USINT/DINT_TO_USINT', _dint_to_usint_ConverterNode);
NodeFactory.AddNodeAsPrototype('IEC Datatypes/Converters/TO_USINT/DT_TO_USINT', _dt_to_usint_ConverterNode);
NodeFactory.AddNodeAsPrototype('IEC Datatypes/Converters/TO_USINT/DWORD_TO_USINT', _dword_to_usint_ConverterNode);
NodeFactory.AddNodeAsPrototype('IEC Datatypes/Converters/TO_USINT/INT_TO_USINT', _int_to_usint_ConverterNode);
NodeFactory.AddNodeAsPrototype('IEC Datatypes/Converters/TO_USINT/LINT_TO_USINT', _lint_to_usint_ConverterNode);
NodeFactory.AddNodeAsPrototype('IEC Datatypes/Converters/TO_USINT/LREAL_TO_USINT', _lreal_to_usint_ConverterNode);
NodeFactory.AddNodeAsPrototype('IEC Datatypes/Converters/TO_USINT/LWORD_TO_USINT', _lword_to_usint_ConverterNode);
NodeFactory.AddNodeAsPrototype('IEC Datatypes/Converters/TO_USINT/REAL_TO_USINT', _real_to_usint_ConverterNode);
NodeFactory.AddNodeAsPrototype('IEC Datatypes/Converters/TO_USINT/SINT_TO_USINT', _sint_to_usint_ConverterNode);
NodeFactory.AddNodeAsPrototype('IEC Datatypes/Converters/TO_USINT/TOD_TO_USINT', _tod_to_usint_ConverterNode);
NodeFactory.AddNodeAsPrototype('IEC Datatypes/Converters/TO_USINT/UDINT_TO_USINT', _udint_to_usint_ConverterNode);
NodeFactory.AddNodeAsPrototype('IEC Datatypes/Converters/TO_USINT/UINT_TO_USINT', _uint_to_usint_ConverterNode);
NodeFactory.AddNodeAsPrototype('IEC Datatypes/Converters/TO_USINT/ULINT_TO_USINT', _ulint_to_usint_ConverterNode);
NodeFactory.AddNodeAsPrototype('IEC Datatypes/Converters/TO_USINT/USINT_TO_USINT', _usint_to_usint_ConverterNode);
NodeFactory.AddNodeAsPrototype('IEC Datatypes/Converters/TO_USINT/WORD_TO_USINT', _word_to_usint_ConverterNode);
NodeFactory.AddNodeAsPrototype('IEC Datatypes/Converters/TO_USINT/STRING_TO_USINT', _string_to_usint_ConverterNode);

// _to_word
NodeFactory.AddNodeAsPrototype('IEC Datatypes/Converters/TO_WORD/BOOL_TO_WORD', _bool_to_word_ConverterNode);
NodeFactory.AddNodeAsPrototype('IEC Datatypes/Converters/TO_WORD/BYTE_TO_WORD', _byte_to_word_ConverterNode);
NodeFactory.AddNodeAsPrototype('IEC Datatypes/Converters/TO_WORD/DINT_TO_WORD', _dint_to_word_ConverterNode);
NodeFactory.AddNodeAsPrototype('IEC Datatypes/Converters/TO_WORD/DT_TO_WORD', _dt_to_word_ConverterNode);
NodeFactory.AddNodeAsPrototype('IEC Datatypes/Converters/TO_WORD/DWORD_TO_WORD', _dword_to_word_ConverterNode);
NodeFactory.AddNodeAsPrototype('IEC Datatypes/Converters/TO_WORD/INT_TO_WORD', _int_to_word_ConverterNode);
NodeFactory.AddNodeAsPrototype('IEC Datatypes/Converters/TO_WORD/LINT_TO_WORD', _lint_to_word_ConverterNode);
NodeFactory.AddNodeAsPrototype('IEC Datatypes/Converters/TO_WORD/LREAL_TO_WORD', _lreal_to_word_ConverterNode);
NodeFactory.AddNodeAsPrototype('IEC Datatypes/Converters/TO_WORD/LWORD_TO_WORD', _lword_to_word_ConverterNode);
NodeFactory.AddNodeAsPrototype('IEC Datatypes/Converters/TO_WORD/REAL_TO_WORD', _real_to_word_ConverterNode);
NodeFactory.AddNodeAsPrototype('IEC Datatypes/Converters/TO_WORD/SINT_TO_WORD', _sint_to_word_ConverterNode);
NodeFactory.AddNodeAsPrototype('IEC Datatypes/Converters/TO_WORD/TOD_TO_WORD', _tod_to_word_ConverterNode);
NodeFactory.AddNodeAsPrototype('IEC Datatypes/Converters/TO_WORD/UDINT_TO_WORD', _udint_to_word_ConverterNode);
NodeFactory.AddNodeAsPrototype('IEC Datatypes/Converters/TO_WORD/UINT_TO_WORD', _uint_to_word_ConverterNode);
NodeFactory.AddNodeAsPrototype('IEC Datatypes/Converters/TO_WORD/ULINT_TO_WORD', _ulint_to_word_ConverterNode);
NodeFactory.AddNodeAsPrototype('IEC Datatypes/Converters/TO_WORD/USINT_TO_WORD', _usint_to_word_ConverterNode);
NodeFactory.AddNodeAsPrototype('IEC Datatypes/Converters/TO_WORD/WORD_TO_WORD', _word_to_word_ConverterNode);
NodeFactory.AddNodeAsPrototype('IEC Datatypes/Converters/TO_WORD/STRING_TO_WORD', _string_to_word_ConverterNode);

// _to_string
NodeFactory.AddNodeAsPrototype('IEC Datatypes/Converters/TO_STRING/BOOL_TO_STRING', _bool_to_string_ConverterNode);
NodeFactory.AddNodeAsPrototype('IEC Datatypes/Converters/TO_STRING/BYTE_TO_STRING', _byte_to_string_ConverterNode);
NodeFactory.AddNodeAsPrototype('IEC Datatypes/Converters/TO_STRING/DINT_TO_STRING', _dint_to_string_ConverterNode);
NodeFactory.AddNodeAsPrototype('IEC Datatypes/Converters/TO_STRING/DT_TO_STRING', _dt_to_string_ConverterNode);
NodeFactory.AddNodeAsPrototype('IEC Datatypes/Converters/TO_STRING/DWORD_TO_STRING', _dword_to_string_ConverterNode);
NodeFactory.AddNodeAsPrototype('IEC Datatypes/Converters/TO_STRING/INT_TO_STRING', _int_to_string_ConverterNode);
NodeFactory.AddNodeAsPrototype('IEC Datatypes/Converters/TO_STRING/LINT_TO_STRING', _lint_to_string_ConverterNode);
NodeFactory.AddNodeAsPrototype('IEC Datatypes/Converters/TO_STRING/LREAL_TO_STRING', _lreal_to_string_ConverterNode);
NodeFactory.AddNodeAsPrototype('IEC Datatypes/Converters/TO_STRING/LWORD_TO_STRING', _lword_to_string_ConverterNode);
NodeFactory.AddNodeAsPrototype('IEC Datatypes/Converters/TO_STRING/REAL_TO_STRING', _real_to_string_ConverterNode);
NodeFactory.AddNodeAsPrototype('IEC Datatypes/Converters/TO_STRING/SINT_TO_STRING', _sint_to_string_ConverterNode);
NodeFactory.AddNodeAsPrototype('IEC Datatypes/Converters/TO_STRING/TOD_TO_STRING', _tod_to_string_ConverterNode);
NodeFactory.AddNodeAsPrototype('IEC Datatypes/Converters/TO_STRING/UDINT_TO_STRING', _udint_to_string_ConverterNode);
NodeFactory.AddNodeAsPrototype('IEC Datatypes/Converters/TO_STRING/UINT_TO_STRING', _uint_to_string_ConverterNode);
NodeFactory.AddNodeAsPrototype('IEC Datatypes/Converters/TO_STRING/ULINT_TO_STRING', _ulint_to_string_ConverterNode);
NodeFactory.AddNodeAsPrototype('IEC Datatypes/Converters/TO_STRING/USINT_TO_STRING', _usint_to_string_ConverterNode);
NodeFactory.AddNodeAsPrototype('IEC Datatypes/Converters/TO_STRING/WORD_TO_STRING', _word_to_string_ConverterNode);
NodeFactory.AddNodeAsPrototype('IEC Datatypes/Converters/TO_STRING/STRING_TO_STRING', _string_to_string_ConverterNode);
END_METHOD

END_FUNCTION_BLOCK

// Node/Converters/ConverterNode
{attribute 'linkalways'} 
{attribute 'no_explicit_call' := 'This FB is a CLASS and must be accessed using methods or properties'}
{attribute 'enable_dynamic_creation'}
FUNCTION_BLOCK FINAL ConverterNode EXTENDS Node
VAR
	in : I_Datatype;
	out : I_Datatype;
	success : _BOOL(false);
END_VAR

METHOD FB_init : BOOL
VAR_INPUT
	bInitRetains : BOOL; // if TRUE, the retain variables are initialized (warm start / cold start)
	bInCopyCode : BOOL;  // if TRUE, the instance afterwards gets moved into the copy code (online change)
	In : I_Datatype;
	Out : I_Datatype;
END_VAR
THIS^.in := In.Clone();
THIS^.out := Out.Clone();

AddInput('in',THIS^.in);
AddOutput('success', THIS^.success);
AddOutput('out', THIS^.out);
END_METHOD

METHOD FB_exit : BOOL
VAR_INPUT
	bInCopyCode : BOOL; // if TRUE, the exit method is called for exiting an instance that is copied afterwards (online change).
END_VAR
IF bInCopyCode THEN
	RETURN;
END_IF

in.Dispose();
out.Dispose();
END_METHOD

METHOD PUBLIC Clone : I_Node
VAR
	pNode : POINTER TO ConverterNode;
END_VAR
pNode := __NEW(ConverterNode(In := THIS^.in, Out := THIS^.out));
Clone := pNode^;
END_METHOD

METHOD PROTECTED OnExecute
VAR
END_VAR
success.Value := in.TryConvertTo_(out);
END_METHOD

END_FUNCTION_BLOCK

// Node/Hardware/HardwareNode
{attribute 'linkalways'} 
{attribute 'no_explicit_call' := 'This FB is a CLASS and must be accessed using methods or properties'}
{attribute 'enable_dynamic_creation'}
{attribute 'hide_all_locals'}
FUNCTION_BLOCK ABSTRACT HardwareNode EXTENDS Node
VAR
END_VAR

METHOD PUBLIC  Clone : I_Node
VAR_INPUT
END_VAR
Clone := THIS^;
// hardware nodes are singletons, so when asked to clone, it instead returns itself.
END_METHOD

METHOD PUBLIC Dispose
VAR_INPUT
END_VAR
// hardware nodes are singletons, so this remains empty as it should not be destroyed.
END_METHOD

END_FUNCTION_BLOCK
